LIN {X 0,Y 439.725,Z 495.084,A -85,B 0,C 180,E1 -9116.585,E2 -9116.585} C_VEL
LIN {X 0,Y 440.208,Z 487.996,A -85,B 0,C 180,E1 -9119.665,E2 -9119.665} C_VEL
LIN {X 0,Y 440.75,Z 482.421,A -85,B 0,C 180,E1 -9122.316,E2 -9122.316} C_VEL
LIN {X 0,Y 441.339,Z 477.409,A -85,B 0,C 180,E1 -9124.979,E2 -9124.979} C_VEL
LIN {X 0,Y 441.446,Z 473.772,A -85,B 0,C 180,E1 -9127.248,E2 -9127.248} C_VEL
LIN {X 0,Y 440.974,Z 470.762,A -85,B 0,C 180,E1 -9129.606,E2 -9129.606} C_VEL
LIN {X 0,Y 440.555,Z 468.312,A -85,B 0,C 180,E1 -9132.068,E2 -9132.068} C_VEL
LIN {X 0,Y 440.223,Z 466.544,A -85,B 0,C 180,E1 -9134.624,E2 -9134.624} C_VEL
LIN {X 0,Y 440.026,Z 465.358,A -85,B 0,C 180,E1 -9137.87,E2 -9137.87} C_VEL
LIN {X 0,Y 439.939,Z 465.185,A -85,B 0,C 180,E1 -9140.283,E2 -9140.283} C_VEL
LIN {X 0,Y 439.949,Z 465.547,A -85,B 0,C 180,E1 -9143.009,E2 -9143.009} C_VEL
LIN {X 0,Y 439.921,Z 466.128,A -85,B 0,C 180,E1 -9144.892,E2 -9144.892} C_VEL
LIN {X 0,Y 439.676,Z 467.615,A -85,B 0,C 180,E1 -9148.164,E2 -9148.164} C_VEL
LIN {X 0,Y 439.382,Z 469.659,A -85,B 0,C 180,E1 -9151.611,E2 -9151.611} C_VEL
LIN {X 0,Y 439.159,Z 471.579,A -85,B 0,C 180,E1 -9154.4,E2 -9154.4} C_VEL
LIN {X 0,Y 438.986,Z 473.84,A -85,B 0,C 180,E1 -9157.404,E2 -9157.404} C_VEL
LIN {X 0,Y 438.856,Z 476.233,A -85,B 0,C 180,E1 -9160.348,E2 -9160.348} C_VEL
LIN {X 0,Y 438.8,Z 479.014,A -85,B 0,C 180,E1 -9163.564,E2 -9163.564} C_VEL
LIN {X 0,Y 442.176,Z 491.192,A -85,B 0,C 180,E1 -9164.187,E2 -9164.187} C_VEL
LIN {X 0,Y 443.053,Z 496.365,A -85,B 0,C 180,E1 -9164.474,E2 -9164.474} C_VEL
LIN {X 0,Y 442.518,Z 508.604,A -85,B 0,C 180,E1 -9165.162,E2 -9165.162} C_VEL
LIN {X 0,Y 441.894,Z 520.706,A -85,B 0,C 180,E1 -9166.046,E2 -9166.046} C_VEL
LIN {X 0,Y 441.212,Z 532.256,A -85,B 0,C 180,E1 -9167.115,E2 -9167.115} C_VEL
LIN {X 0,Y 440.547,Z 542.238,A -85,B 0,C 180,E1 -9168.264,E2 -9168.264} C_VEL
LIN {X 0,Y 439.943,Z 551.84,A -85,B 0,C 180,E1 -9169.647,E2 -9169.647} C_VEL
LIN {X 0,Y 439.48,Z 559.568,A -85,B 0,C 180,E1 -9171.03,E2 -9171.03} C_VEL
LIN {X 0,Y 439.157,Z 564.797,A -85,B 0,C 180,E1 -9172.182,E2 -9172.182} C_VEL
LIN {X 0,Y 438.905,Z 569.893,A -85,B 0,C 180,E1 -9173.564,E2 -9173.564} C_VEL
LIN {X 0,Y 438.658,Z 573.844,A -85,B 0,C 180,E1 -9174.945,E2 -9174.945} C_VEL
LIN {X 0,Y 438.567,Z 576.739,A -85,B 0,C 180,E1 -9176.325,E2 -9176.325} C_VEL
LIN {X 0,Y 438.497,Z 578.115,A -85,B 0,C 180,E1 -9177.244,E2 -9177.244} C_VEL
LIN {X 0,Y 438.465,Z 579.07,A -85,B 0,C 180,E1 -9178.163,E2 -9178.163} C_VEL
LIN {X 0,Y 438.368,Z 579.638,A -85,B 0,C 180,E1 -9179.082,E2 -9179.082} C_VEL
LIN {X 0,Y 438.338,Z 579.807,A -85,B 0,C 180,E1 -9180,E2 -9180} C_VEL
LIN {X 0,Y 438.368,Z 579.532,A -85,B 0,C 180,E1 -9180.919,E2 -9180.919} C_VEL
LIN {X 0,Y 438.416,Z 578.858,A -85,B 0,C 180,E1 -9181.837,E2 -9181.837} C_VEL
LIN {X 0,Y 438.473,Z 577.791,A -85,B 0,C 180,E1 -9182.756,E2 -9182.756} C_VEL
LIN {X 0,Y 438.55,Z 576.305,A -85,B 0,C 180,E1 -9183.676,E2 -9183.676} C_VEL
LIN {X 0,Y 438.55,Z 573.247,A -85,B 0,C 180,E1 -9185.057,E2 -9185.057} C_VEL
LIN {X 0,Y 438.843,Z 569.115,A -85,B 0,C 180,E1 -9186.437,E2 -9186.437} C_VEL
LIN {X 0,Y 439.061,Z 562.782,A -85,B 0,C 180,E1 -9188.052,E2 -9188.052} C_VEL
LIN {X 0,Y 439.463,Z 555.889,A -85,B 0,C 180,E1 -9189.435,E2 -9189.435} C_VEL
LIN {X 0,Y 439.838,Z 548.87,A -85,B 0,C 180,E1 -9190.589,E2 -9190.589} C_VEL
LIN {X 0,Y 440.275,Z 540.435,A -85,B 0,C 180,E1 -9191.743,E2 -9191.743} C_VEL
LIN {X 0,Y 440.958,Z 530.059,A -85,B 0,C 180,E1 -9192.893,E2 -9192.893} C_VEL
LIN {X 0,Y 441.475,Z 518.456,A -85,B 0,C 180,E1 -9193.933,E2 -9193.933} C_VEL
LIN {X 0,Y 441.995,Z 507.041,A -85,B 0,C 180,E1 -9194.739,E2 -9194.739} C_VEL
LIN {X 0,Y 442.48,Z 495.475,A -85,B 0,C 180,E1 -9195.37,E2 -9195.37} C_VEL
LIN {X 0,Y 441.325,Z 488.815,A -85,B 0,C 180,E1 -9195.708,E2 -9195.708} C_VEL
LIN {X 0,Y 438.492,Z 476.161,A -85,B 0,C 180,E1 -9196.254,E2 -9196.254} C_VEL
LIN {X 0,Y 438.499,Z 472.466,A -85,B 0,C 180,E1 -9199.669,E2 -9199.669} C_VEL
LIN {X 0,Y 438.541,Z 469.335,A -85,B 0,C 180,E1 -9202.621,E2 -9202.621} C_VEL
LIN {X 0,Y 438.665,Z 465.591,A -85,B 0,C 180,E1 -9206.208,E2 -9206.208} C_VEL
LIN {X 0,Y 438.668,Z 463.019,A -85,B 0,C 180,E1 -9208.727,E2 -9208.727} C_VEL
LIN {X 0,Y 438.728,Z 461.844,A -85,B 0,C 180,E1 -9210.114,E2 -9210.114} C_VEL
LIN {X 0,Y 439.044,Z 461.798,A -85,B 0,C 180,E1 -9212.974,E2 -9212.974} C_VEL
LIN {X 0,Y 439.311,Z 461.762,A -85,B 0,C 180,E1 -9215.324,E2 -9215.324} C_VEL
LIN {X 0,Y 439.378,Z 461.756,A -85,B 0,C 180,E1 -9218.596,E2 -9218.596} C_VEL
LIN {X 0,Y 439.394,Z 461.749,A -85,B 0,C 180,E1 -9221.257,E2 -9221.257} C_VEL
LIN {X 0,Y 439.41,Z 461.75,A -85,B 0,C 180,E1 -9224.729,E2 -9224.729} C_VEL
LIN {X 0,Y 439.4,Z 461.753,A -85,B 0,C 180,E1 -9227.796,E2 -9227.796} C_VEL
LIN {X 0,Y 439.441,Z 461.747,A -85,B 0,C 180,E1 -9230.229,E2 -9230.229} C_VEL
LIN {X 0,Y 439.378,Z 461.753,A -85,B 0,C 180,E1 -9233.713,E2 -9233.713} C_VEL
LIN {X 0,Y 439.377,Z 461.754,A -85,B 0,C 180,E1 -9237.054,E2 -9237.054} C_VEL
LIN {X 0,Y 439.387,Z 461.753,A -85,B 0,C 180,E1 -9240.274,E2 -9240.274} C_VEL
LIN {X 0,Y 439.433,Z 461.747,A -85,B 0,C 180,E1 -9243.396,E2 -9243.396} C_VEL
LIN {X 0,Y 439.389,Z 461.753,A -85,B 0,C 180,E1 -9246.43,E2 -9246.43} C_VEL
LIN {X 0,Y 439.393,Z 461.752,A -85,B 0,C 180,E1 -9249.397,E2 -9249.397} C_VEL
LIN {X 0,Y 439.431,Z 461.748,A -85,B 0,C 180,E1 -9252.309,E2 -9252.309} C_VEL
LIN {X 0,Y 439.453,Z 461.744,A -85,B 0,C 180,E1 -9255.174,E2 -9255.174} C_VEL
LIN {X 0,Y 439.489,Z 461.742,A -85,B 0,C 180,E1 -9258.001,E2 -9258.001} C_VEL
LIN {X 0,Y 439.553,Z 461.735,A -85,B 0,C 180,E1 -9261.726,E2 -9261.726} C_VEL
LIN {X 0,Y 439.626,Z 461.724,A -85,B 0,C 180,E1 -9264.496,E2 -9264.496} C_VEL
LIN {X 0,Y 439.573,Z 461.729,A -85,B 0,C 180,E1 -9266.99,E2 -9266.99} C_VEL
LIN {X 0,Y 439.046,Z 461.796,A -85,B 0,C 180,E1 -9267.755,E2 -9267.755} C_VEL
LIN {X 0,Y 436.22,Z 462.147,A -85,B 0,C 180,E1 -9268.998,E2 -9268.998} C_VEL
LIN {X 0,Y 433.737,Z 462.459,A -85,B 0,C 180,E1 -9270.001,E2 -9270.001} C_VEL
LIN {X 0,Y 432.661,Z 462.589,A -85,B 0,C 180,E1 -9270.777,E2 -9270.777} C_VEL
LIN {X 0,Y 432.574,Z 462.599,A -85,B 0,C 180,E1 -9271.04,E2 -9271.04} C_VEL
LIN {X 0,Y 432.597,Z 462.597,A -85,B 0,C 180,E1 -9272.794,E2 -9272.794} C_VEL
LIN {X 0,Y 432.591,Z 462.602,A -85,B 0,C 180,E1 -9275.594,E2 -9275.594} C_VEL
LIN {X 0,Y 432.469,Z 462.617,A -85,B 0,C 180,E1 -9278.41,E2 -9278.41} C_VEL
LIN {X 0,Y 432.465,Z 462.617,A -85,B 0,C 180,E1 -9282.196,E2 -9282.196} C_VEL
LIN {X 0,Y 432.436,Z 462.62,A -85,B 0,C 180,E1 -9286.039,E2 -9286.039} C_VEL
LIN {X 0,Y 432.392,Z 462.626,A -85,B 0,C 180,E1 -9289.485,E2 -9289.485} C_VEL
LIN {X 0,Y 432.323,Z 462.632,A -85,B 0,C 180,E1 -9292.964,E2 -9292.964} C_VEL
LIN {X 0,Y 432.366,Z 462.629,A -85,B 0,C 180,E1 -9296.032,E2 -9296.032} C_VEL
LIN {X 0,Y 432.348,Z 462.629,A -85,B 0,C 180,E1 -9299.187,E2 -9299.187} C_VEL
LIN {X 0,Y 432.328,Z 462.633,A -85,B 0,C 180,E1 -9302.443,E2 -9302.443} C_VEL
LIN {X 0,Y 432.35,Z 462.63,A -85,B 0,C 180,E1 -9305.632,E2 -9305.632} C_VEL
LIN {X 0,Y 432.357,Z 462.625,A -85,B 0,C 180,E1 -9308.716,E2 -9308.716} C_VEL
LIN {X 0,Y 432.338,Z 462.632,A -85,B 0,C 180,E1 -9311.797,E2 -9311.797} C_VEL
LIN {X 0,Y 432.338,Z 462.632,A -85,B 0,C 180,E1 -9314.347,E2 -9314.347} C_VEL
LIN {X 0,Y 432.329,Z 462.632,A -85,B 0,C 180,E1 -9317.015,E2 -9317.015} C_VEL
LIN {X 0,Y 432.338,Z 462.634,A -85,B 0,C 180,E1 -9319.82,E2 -9319.82} C_VEL
LIN {X 0,Y 432.303,Z 462.634,A -85,B 0,C 180,E1 -9323.021,E2 -9323.021} C_VEL
LIN {X 0,Y 432.247,Z 462.645,A -85,B 0,C 180,E1 -9325.314,E2 -9325.314} C_VEL
LIN {X 0,Y 432.019,Z 462.674,A -85,B 0,C 180,E1 -9327.772,E2 -9327.772} C_VEL
LIN {X 0,Y 431.603,Z 462.726,A -85,B 0,C 180,E1 -9330.757,E2 -9330.757} C_VEL
LIN {X 0,Y 431.523,Z 462.84,A -85,B 0,C 180,E1 -9331.815,E2 -9331.815} C_VEL
LIN {X 0,Y 431.446,Z 466.378,A -85,B 0,C 180,E1 -9334.942,E2 -9334.942} C_VEL
LIN {X 0,Y 431.436,Z 470.05,A -85,B 0,C 180,E1 -9338.206,E2 -9338.206} C_VEL
LIN {X 0,Y 431.423,Z 473.199,A -85,B 0,C 180,E1 -9340.985,E2 -9340.985} C_VEL
LIN {X 0,Y 431.386,Z 476.277,A -85,B 0,C 180,E1 -9343.637,E2 -9343.637} C_VEL
LIN {X 0,Y 434.162,Z 488.766,A -85,B 0,C 180,E1 -9344.163,E2 -9344.163} C_VEL
LIN {X 0,Y 435.505,Z 496.504,A -85,B 0,C 180,E1 -9344.567,E2 -9344.567} C_VEL
LIN {X 0,Y 434.983,Z 508.593,A -85,B 0,C 180,E1 -9345.257,E2 -9345.257} C_VEL
LIN {X 0,Y 434.531,Z 519.197,A -85,B 0,C 180,E1 -9346.032,E2 -9346.032} C_VEL
LIN {X 0,Y 433.994,Z 529.992,A -85,B 0,C 180,E1 -9347.015,E2 -9347.015} C_VEL
LIN {X 0,Y 433.343,Z 539.442,A -85,B 0,C 180,E1 -9348.066,E2 -9348.066} C_VEL
LIN {X 0,Y 432.877,Z 548.128,A -85,B 0,C 180,E1 -9349.239,E2 -9349.239} C_VEL
LIN {X 0,Y 432.357,Z 556.622,A -85,B 0,C 180,E1 -9350.645,E2 -9350.645} C_VEL
LIN {X 0,Y 431.951,Z 563.423,A -85,B 0,C 180,E1 -9352.05,E2 -9352.05} C_VEL
LIN {X 0,Y 431.779,Z 568.864,A -85,B 0,C 180,E1 -9353.457,E2 -9353.457} C_VEL
LIN {X 0,Y 431.474,Z 573.12,A -85,B 0,C 180,E1 -9354.86,E2 -9354.86} C_VEL
LIN {X 0,Y 431.472,Z 576.287,A -85,B 0,C 180,E1 -9356.264,E2 -9356.264} C_VEL
LIN {X 0,Y 431.394,Z 577.87,A -85,B 0,C 180,E1 -9357.198,E2 -9357.198} C_VEL
LIN {X 0,Y 431.321,Z 578.99,A -85,B 0,C 180,E1 -9358.132,E2 -9358.132} C_VEL
LIN {X 0,Y 431.279,Z 580.034,A -85,B 0,C 180,E1 -9360,E2 -9360} C_VEL
LIN {X 0,Y 431.31,Z 579.937,A -85,B 0,C 180,E1 -9360.933,E2 -9360.933} C_VEL
LIN {X 0,Y 431.393,Z 579.41,A -85,B 0,C 180,E1 -9361.867,E2 -9361.867} C_VEL
LIN {X 0,Y 431.425,Z 578.499,A -85,B 0,C 180,E1 -9362.801,E2 -9362.801} C_VEL
LIN {X 0,Y 431.514,Z 577.184,A -85,B 0,C 180,E1 -9363.735,E2 -9363.735} C_VEL
LIN {X 0,Y 431.57,Z 574.377,A -85,B 0,C 180,E1 -9365.138,E2 -9365.138} C_VEL
LIN {X 0,Y 431.861,Z 570.513,A -85,B 0,C 180,E1 -9366.541,E2 -9366.541} C_VEL
LIN {X 0,Y 432.098,Z 565.493,A -85,B 0,C 180,E1 -9367.946,E2 -9367.946} C_VEL
LIN {X 0,Y 432.62,Z 557.957,A -85,B 0,C 180,E1 -9369.585,E2 -9369.585} C_VEL
LIN {X 0,Y 433.15,Z 549.779,A -85,B 0,C 180,E1 -9370.99,E2 -9370.99} C_VEL
LIN {X 0,Y 433.839,Z 539.573,A -85,B 0,C 180,E1 -9372.394,E2 -9372.394} C_VEL
LIN {X 0,Y 434.525,Z 529.567,A -85,B 0,C 180,E1 -9373.499,E2 -9373.499} C_VEL
LIN {X 0,Y 435.124,Z 518.422,A -85,B 0,C 180,E1 -9374.498,E2 -9374.498} C_VEL
LIN {X 0,Y 435.834,Z 506.924,A -85,B 0,C 180,E1 -9375.311,E2 -9375.311} C_VEL
LIN {X 0,Y 436.243,Z 496.479,A -85,B 0,C 180,E1 -9375.895,E2 -9375.895} C_VEL
LIN {X 0,Y 433.618,Z 485.375,A -85,B 0,C 180,E1 -9376.517,E2 -9376.517} C_VEL
LIN {X 0,Y 431.621,Z 478.702,A -85,B 0,C 180,E1 -9376.883,E2 -9376.883} C_VEL
LIN {X 0,Y 431.656,Z 475.198,A -85,B 0,C 180,E1 -9379.993,E2 -9379.993} C_VEL
LIN {X 0,Y 431.671,Z 471.756,A -85,B 0,C 180,E1 -9383.001,E2 -9383.001} C_VEL
LIN {X 0,Y 431.767,Z 467.645,A -85,B 0,C 180,E1 -9386.459,E2 -9386.459} C_VEL
LIN {X 0,Y 431.733,Z 464.394,A -85,B 0,C 180,E1 -9389.233,E2 -9389.233} C_VEL
LIN {X 0,Y 431.727,Z 462.935,A -85,B 0,C 180,E1 -9390.37,E2 -9390.37} C_VEL
LIN {X 0,Y 432.045,Z 462.672,A -85,B 0,C 180,E1 -9392.466,E2 -9392.466} C_VEL
LIN {X 0,Y 432.314,Z 462.636,A -85,B 0,C 180,E1 -9395.626,E2 -9395.626} C_VEL
LIN {X 0,Y 432.35,Z 462.63,A -85,B 0,C 180,E1 -9398.716,E2 -9398.716} C_VEL
LIN {X 0,Y 432.337,Z 462.632,A -85,B 0,C 180,E1 -9401.797,E2 -9401.797} C_VEL
LIN {X 0,Y 432.343,Z 462.633,A -85,B 0,C 180,E1 -9404.346,E2 -9404.346} C_VEL
LIN {X 0,Y 432.374,Z 462.673,A -85,B 0,C 180,E1 -9408.129,E2 -9408.129} C_VEL
LIN {X 0,Y 433.449,Z 468.757,A -85,B 0,C 180,E1 -9411.103,E2 -9411.103} C_VEL
LIN {X 0,Y 434.2,Z 473.235,A -85,B 0,C 180,E1 -9413.21,E2 -9413.21} C_VEL
LIN {X 0,Y 434.325,Z 477.103,A -85,B 0,C 180,E1 -9414.939,E2 -9414.939} C_VEL
LIN {X 0,Y 433.664,Z 484.792,A -85,B 0,C 180,E1 -9418.217,E2 -9418.217} C_VEL
LIN {X 0,Y 433.229,Z 491.9,A -85,B 0,C 180,E1 -9421.165,E2 -9421.165} C_VEL
LIN {X 0,Y 432.674,Z 500.183,A -85,B 0,C 180,E1 -9424.504,E2 -9424.504} C_VEL
LIN {X 0,Y 432.218,Z 509.175,A -85,B 0,C 180,E1 -9428.038,E2 -9428.038} C_VEL
LIN {X 0,Y 431.858,Z 518.157,A -85,B 0,C 180,E1 -9431.498,E2 -9431.498} C_VEL
LIN {X 0,Y 431.738,Z 523.3,A -85,B 0,C 180,E1 -9433.454,E2 -9433.454} C_VEL
LIN {X 0,Y 433.768,Z 537.812,A -85,B 0,C 180,E1 -9433.992,E2 -9433.992} C_VEL
LIN {X 0,Y 435.049,Z 549.897,A -85,B 0,C 180,E1 -9434.601,E2 -9434.601} C_VEL
LIN {X 0,Y 434.387,Z 562.251,A -85,B 0,C 180,E1 -9435.357,E2 -9435.357} C_VEL
LIN {X 0,Y 433.768,Z 573.811,A -85,B 0,C 180,E1 -9436.268,E2 -9436.268} C_VEL
LIN {X 0,Y 433.153,Z 584.686,A -85,B 0,C 180,E1 -9437.347,E2 -9437.347} C_VEL
LIN {X 0,Y 432.586,Z 594.309,A -85,B 0,C 180,E1 -9438.52,E2 -9438.52} C_VEL
LIN {X 0,Y 432.077,Z 602.225,A -85,B 0,C 180,E1 -9439.693,E2 -9439.693} C_VEL
LIN {X 0,Y 431.724,Z 609.974,A -85,B 0,C 180,E1 -9441.103,E2 -9441.103} C_VEL
LIN {X 0,Y 431.465,Z 616.192,A -85,B 0,C 180,E1 -9442.512,E2 -9442.512} C_VEL
LIN {X 0,Y 431.299,Z 621.368,A -85,B 0,C 180,E1 -9444.002,E2 -9444.002} C_VEL
LIN {X 0,Y 431.289,Z 624.889,A -85,B 0,C 180,E1 -9445.327,E2 -9445.327} C_VEL
LIN {X 0,Y 431.238,Z 626.819,A -85,B 0,C 180,E1 -9446.262,E2 -9446.262} C_VEL
LIN {X 0,Y 431.318,Z 628.308,A -85,B 0,C 180,E1 -9447.198,E2 -9447.198} C_VEL
LIN {X 0,Y 431.285,Z 629.327,A -85,B 0,C 180,E1 -9448.132,E2 -9448.132} C_VEL
LIN {X 0,Y 431.289,Z 629.944,A -85,B 0,C 180,E1 -9449.066,E2 -9449.066} C_VEL
LIN {X 0,Y 431.277,Z 630.156,A -85,B 0,C 180,E1 -9450,E2 -9450} C_VEL
LIN {X 0,Y 431.276,Z 629.931,A -85,B 0,C 180,E1 -9450.934,E2 -9450.934} C_VEL
LIN {X 0,Y 431.287,Z 629.272,A -85,B 0,C 180,E1 -9451.868,E2 -9451.868} C_VEL
LIN {X 0,Y 431.326,Z 628.209,A -85,B 0,C 180,E1 -9452.802,E2 -9452.802} C_VEL
LIN {X 0,Y 431.245,Z 626.725,A -85,B 0,C 180,E1 -9453.738,E2 -9453.738} C_VEL
LIN {X 0,Y 431.329,Z 623.63,A -85,B 0,C 180,E1 -9455.142,E2 -9455.142} C_VEL
LIN {X 0,Y 431.376,Z 619.459,A -85,B 0,C 180,E1 -9456.549,E2 -9456.549} C_VEL
LIN {X 0,Y 431.6,Z 613.079,A -85,B 0,C 180,E1 -9458.191,E2 -9458.191} C_VEL
LIN {X 0,Y 431.891,Z 606.139,A -85,B 0,C 180,E1 -9459.602,E2 -9459.602} C_VEL
LIN {X 0,Y 432.365,Z 597.585,A -85,B 0,C 180,E1 -9461.011,E2 -9461.011} C_VEL
LIN {X 0,Y 432.9,Z 588.865,A -85,B 0,C 180,E1 -9462.184,E2 -9462.184} C_VEL
LIN {X 0,Y 433.491,Z 578.875,A -85,B 0,C 180,E1 -9463.292,E2 -9463.292} C_VEL
LIN {X 0,Y 434.191,Z 567.869,A -85,B 0,C 180,E1 -9464.291,E2 -9464.291} C_VEL
LIN {X 0,Y 434.922,Z 556.771,A -85,B 0,C 180,E1 -9465.104,E2 -9465.104} C_VEL
LIN {X 0,Y 435.135,Z 547.972,A -85,B 0,C 180,E1 -9465.636,E2 -9465.636} C_VEL
LIN {X 0,Y 433.873,Z 534.203,A -85,B 0,C 180,E1 -9466.359,E2 -9466.359} C_VEL
LIN {X 0,Y 431.663,Z 520.58,A -85,B 0,C 180,E1 -9466.942,E2 -9466.942} C_VEL
LIN {X 0,Y 431.956,Z 511.211,A -85,B 0,C 180,E1 -9470.476,E2 -9470.476} C_VEL
LIN {X 0,Y 432.235,Z 503.577,A -85,B 0,C 180,E1 -9473.476,E2 -9473.476} C_VEL
LIN {X 0,Y 432.696,Z 495.781,A -85,B 0,C 180,E1 -9476.705,E2 -9476.705} C_VEL
LIN {X 0,Y 433.19,Z 489.162,A -85,B 0,C 180,E1 -9479.658,E2 -9479.658} C_VEL
LIN {X 0,Y 433.75,Z 483.692,A -85,B 0,C 180,E1 -9482.323,E2 -9482.323} C_VEL
LIN {X 0,Y 434.28,Z 479.633,A -85,B 0,C 180,E1 -9484.5,E2 -9484.5} C_VEL
LIN {X 0,Y 434.482,Z 475.964,A -85,B 0,C 180,E1 -9486.762,E2 -9486.762} C_VEL
LIN {X 0,Y 434.141,Z 472.803,A -85,B 0,C 180,E1 -9489.15,E2 -9489.15} C_VEL
LIN {X 0,Y 433.676,Z 470.093,A -85,B 0,C 180,E1 -9491.801,E2 -9491.801} C_VEL
LIN {X 0,Y 433.307,Z 468.189,A -85,B 0,C 180,E1 -9494.467,E2 -9494.467} C_VEL
LIN {X 0,Y 433.135,Z 467.082,A -85,B 0,C 180,E1 -9497.04,E2 -9497.04} C_VEL
LIN {X 0,Y 432.998,Z 466.649,A -85,B 0,C 180,E1 -9499.717,E2 -9499.717} C_VEL
LIN {X 0,Y 432.987,Z 466.95,A -85,B 0,C 180,E1 -9503.09,E2 -9503.09} C_VEL
LIN {X 0,Y 432.852,Z 467.822,A -85,B 0,C 180,E1 -9505.901,E2 -9505.901} C_VEL
LIN {X 0,Y 432.637,Z 469.107,A -85,B 0,C 180,E1 -9508.679,E2 -9508.679} C_VEL
LIN {X 0,Y 432.334,Z 470.952,A -85,B 0,C 180,E1 -9511.873,E2 -9511.873} C_VEL
LIN {X 0,Y 432.116,Z 473.054,A -85,B 0,C 180,E1 -9514.984,E2 -9514.984} C_VEL
LIN {X 0,Y 431.942,Z 475.336,A -85,B 0,C 180,E1 -9518.038,E2 -9518.038} C_VEL
LIN {X 0,Y 431.869,Z 477.718,A -85,B 0,C 180,E1 -9521.006,E2 -9521.006} C_VEL
LIN {X 0,Y 431.796,Z 479.791,A -85,B 0,C 180,E1 -9523.228,E2 -9523.228} C_VEL
LIN {X 0,Y 435.363,Z 492.152,A -85,B 0,C 180,E1 -9523.9,E2 -9523.9} C_VEL
LIN {X 0,Y 436.316,Z 497.847,A -85,B 0,C 180,E1 -9524.228,E2 -9524.228} C_VEL
LIN {X 0,Y 435.766,Z 509.831,A -85,B 0,C 180,E1 -9524.926,E2 -9524.926} C_VEL
LIN {X 0,Y 435.076,Z 521.704,A -85,B 0,C 180,E1 -9525.822,E2 -9525.822} C_VEL
LIN {X 0,Y 434.341,Z 533.084,A -85,B 0,C 180,E1 -9526.907,E2 -9526.907} C_VEL
LIN {X 0,Y 433.634,Z 542.93,A -85,B 0,C 180,E1 -9528.075,E2 -9528.075} C_VEL
LIN {X 0,Y 432.986,Z 552.482,A -85,B 0,C 180,E1 -9529.479,E2 -9529.479} C_VEL
LIN {X 0,Y 432.502,Z 560.172,A -85,B 0,C 180,E1 -9530.884,E2 -9530.884} C_VEL
LIN {X 0,Y 432.004,Z 567.193,A -85,B 0,C 180,E1 -9532.522,E2 -9532.522} C_VEL
LIN {X 0,Y 431.74,Z 571.862,A -85,B 0,C 180,E1 -9533.926,E2 -9533.926} C_VEL
LIN {X 0,Y 431.63,Z 575.41,A -85,B 0,C 180,E1 -9535.33,E2 -9535.33} C_VEL
LIN {X 0,Y 431.516,Z 577.232,A -85,B 0,C 180,E1 -9536.265,E2 -9536.265} C_VEL
LIN {X 0,Y 431.425,Z 578.584,A -85,B 0,C 180,E1 -9537.199,E2 -9537.199} C_VEL
LIN {X 0,Y 431.409,Z 579.522,A -85,B 0,C 180,E1 -9538.133,E2 -9538.133} C_VEL
LIN {X 0,Y 431.31,Z 580.076,A -85,B 0,C 180,E1 -9539.067,E2 -9539.067} C_VEL
LIN {X 0,Y 431.278,Z 580.227,A -85,B 0,C 180,E1 -9540,E2 -9540} C_VEL
LIN {X 0,Y 431.292,Z 579.934,A -85,B 0,C 180,E1 -9540.934,E2 -9540.934} C_VEL
LIN {X 0,Y 431.334,Z 579.244,A -85,B 0,C 180,E1 -9541.868,E2 -9541.868} C_VEL
LIN {X 0,Y 431.403,Z 578.161,A -85,B 0,C 180,E1 -9542.802,E2 -9542.802} C_VEL
LIN {X 0,Y 431.473,Z 576.648,A -85,B 0,C 180,E1 -9543.736,E2 -9543.736} C_VEL
LIN {X 0,Y 431.485,Z 573.556,A -85,B 0,C 180,E1 -9545.14,E2 -9545.14} C_VEL
LIN {X 0,Y 431.785,Z 569.382,A -85,B 0,C 180,E1 -9546.543,E2 -9546.543} C_VEL
LIN {X 0,Y 432.011,Z 562.998,A -85,B 0,C 180,E1 -9548.184,E2 -9548.184} C_VEL
LIN {X 0,Y 432.455,Z 556.058,A -85,B 0,C 180,E1 -9549.589,E2 -9549.589} C_VEL
LIN {X 0,Y 432.86,Z 548.987,A -85,B 0,C 180,E1 -9550.762,E2 -9550.762} C_VEL
LIN {X 0,Y 433.304,Z 540.485,A -85,B 0,C 180,E1 -9551.935,E2 -9551.935} C_VEL
LIN {X 0,Y 434.031,Z 530.023,A -85,B 0,C 180,E1 -9553.103,E2 -9553.103} C_VEL
LIN {X 0,Y 434.581,Z 518.343,A -85,B 0,C 180,E1 -9554.159,E2 -9554.159} C_VEL
LIN {X 0,Y 435.138,Z 506.769,A -85,B 0,C 180,E1 -9554.977,E2 -9554.977} C_VEL
LIN {X 0,Y 435.504,Z 495.064,A -85,B 0,C 180,E1 -9555.623,E2 -9555.623} C_VEL
LIN {X 0,Y 432.548,Z 481.624,A -85,B 0,C 180,E1 -9556.281,E2 -9556.281} C_VEL
LIN {X 0,Y 431.414,Z 476.484,A -85,B 0,C 180,E1 -9556.504,E2 -9556.504} C_VEL
LIN {X 0,Y 431.42,Z 472.725,A -85,B 0,C 180,E1 -9560.005,E2 -9560.005} C_VEL
LIN {X 0,Y 431.498,Z 469.551,A -85,B 0,C 180,E1 -9563.011,E2 -9563.011} C_VEL
LIN {X 0,Y 431.602,Z 466.032,A -85,B 0,C 180,E1 -9566.415,E2 -9566.415} C_VEL
LIN {X 0,Y 431.614,Z 463.167,A -85,B 0,C 180,E1 -9569.242,E2 -9569.242} C_VEL
LIN {X 0,Y 431.704,Z 462.718,A -85,B 0,C 180,E1 -9570.365,E2 -9570.365} C_VEL
LIN {X 0,Y 432.06,Z 462.667,A -85,B 0,C 180,E1 -9573.577,E2 -9573.577} C_VEL
LIN {X 0,Y 432.27,Z 462.64,A -85,B 0,C 180,E1 -9575.825,E2 -9575.825} C_VEL
LIN {X 0,Y 432.341,Z 462.632,A -85,B 0,C 180,E1 -9578.714,E2 -9578.714} C_VEL
LIN {X 0,Y 432.339,Z 462.63,A -85,B 0,C 180,E1 -9581.797,E2 -9581.797} C_VEL
LIN {X 0,Y 432.345,Z 462.631,A -85,B 0,C 180,E1 -9584.347,E2 -9584.347} C_VEL
LIN {X 0,Y 432.324,Z 462.633,A -85,B 0,C 180,E1 -9587.016,E2 -9587.016} C_VEL
LIN {X 0,Y 432.345,Z 462.63,A -85,B 0,C 180,E1 -9589.82,E2 -9589.82} C_VEL
LIN {X 0,Y 432.315,Z 462.631,A -85,B 0,C 180,E1 -9593.023,E2 -9593.023} C_VEL
LIN {X 0,Y 432.364,Z 462.631,A -85,B 0,C 180,E1 -9595.997,E2 -9595.997} C_VEL
LIN {X 0,Y 432.352,Z 462.63,A -85,B 0,C 180,E1 -9599.49,E2 -9599.49} C_VEL
LIN {X 0,Y 432.395,Z 462.623,A -85,B 0,C 180,E1 -9602.928,E2 -9602.928} C_VEL
LIN {X 0,Y 432.373,Z 462.629,A -85,B 0,C 180,E1 -9606.023,E2 -9606.023} C_VEL
LIN {X 0,Y 432.355,Z 462.628,A -85,B 0,C 180,E1 -9609.046,E2 -9609.046} C_VEL
LIN {X 0,Y 432.379,Z 462.626,A -85,B 0,C 180,E1 -9612.011,E2 -9612.011} C_VEL
LIN {X 0,Y 432.401,Z 462.623,A -85,B 0,C 180,E1 -9614.927,E2 -9614.927} C_VEL
LIN {X 0,Y 432.465,Z 462.616,A -85,B 0,C 180,E1 -9617.804,E2 -9617.804} C_VEL
LIN {X 0,Y 432.497,Z 462.612,A -85,B 0,C 180,E1 -9621.59,E2 -9621.59} C_VEL
LIN {X 0,Y 432.602,Z 462.599,A -85,B 0,C 180,E1 -9624.406,E2 -9624.406} C_VEL
LIN {X 0,Y 432.609,Z 462.599,A -85,B 0,C 180,E1 -9628.138,E2 -9628.138} C_VEL
LIN {X 0,Y 432.738,Z 462.584,A -85,B 0,C 180,E1 -9630,E2 -9630} C_VEL
LIN {X 0,Y 432.574,Z 462.599,A -85,B 0,C 180,E1 -9631.04,E2 -9631.04} C_VEL
LIN {X 0,Y 431.875,Z 462.691,A -85,B 0,C 180,E1 -9631.817,E2 -9631.817} C_VEL
LIN {X 0,Y 428.911,Z 463.056,A -85,B 0,C 180,E1 -9633.076,E2 -9633.076} C_VEL
LIN {X 0,Y 426.456,Z 463.365,A -85,B 0,C 180,E1 -9634.093,E2 -9634.093} C_VEL
LIN {X 0,Y 425.473,Z 463.485,A -85,B 0,C 180,E1 -9634.88,E2 -9634.88} C_VEL
LIN {X 0,Y 425.432,Z 463.49,A -85,B 0,C 180,E1 -9635.147,E2 -9635.147} C_VEL
LIN {X 0,Y 425.484,Z 463.486,A -85,B 0,C 180,E1 -9637.663,E2 -9637.663} C_VEL
LIN {X 0,Y 425.37,Z 463.5,A -85,B 0,C 180,E1 -9640.471,E2 -9640.471} C_VEL
LIN {X 0,Y 425.371,Z 463.497,A -85,B 0,C 180,E1 -9643.374,E2 -9643.374} C_VEL
LIN {X 0,Y 425.367,Z 463.499,A -85,B 0,C 180,E1 -9646.605,E2 -9646.605} C_VEL
LIN {X 0,Y 425.334,Z 463.505,A -85,B 0,C 180,E1 -9649.636,E2 -9649.636} C_VEL
LIN {X 0,Y 425.293,Z 463.51,A -85,B 0,C 180,E1 -9652.339,E2 -9652.339} C_VEL
LIN {X 0,Y 425.296,Z 463.508,A -85,B 0,C 180,E1 -9655.445,E2 -9655.445} C_VEL
LIN {X 0,Y 425.353,Z 463.502,A -85,B 0,C 180,E1 -9657.558,E2 -9657.558} C_VEL
LIN {X 0,Y 425.293,Z 463.508,A -85,B 0,C 180,E1 -9660.816,E2 -9660.816} C_VEL
LIN {X 0,Y 425.317,Z 463.507,A -85,B 0,C 180,E1 -9664.288,E2 -9664.288} C_VEL
LIN {X 0,Y 425.29,Z 463.511,A -85,B 0,C 180,E1 -9667.693,E2 -9667.693} C_VEL
LIN {X 0,Y 425.288,Z 463.508,A -85,B 0,C 180,E1 -9670.521,E2 -9670.521} C_VEL
LIN {X 0,Y 425.262,Z 463.514,A -85,B 0,C 180,E1 -9673.351,E2 -9673.351} C_VEL
LIN {X 0,Y 425.268,Z 463.511,A -85,B 0,C 180,E1 -9676.648,E2 -9676.648} C_VEL
LIN {X 0,Y 425.291,Z 463.512,A -85,B 0,C 180,E1 -9679.873,E2 -9679.873} C_VEL
LIN {X 0,Y 425.278,Z 463.508,A -85,B 0,C 180,E1 -9682.489,E2 -9682.489} C_VEL
LIN {X 0,Y 425.253,Z 463.513,A -85,B 0,C 180,E1 -9684.659,E2 -9684.659} C_VEL
LIN {X 0,Y 425.003,Z 463.548,A -85,B 0,C 180,E1 -9687.496,E2 -9687.496} C_VEL
LIN {X 0,Y 424.507,Z 463.612,A -85,B 0,C 180,E1 -9691.337,E2 -9691.337} C_VEL
LIN {X 0,Y 424.444,Z 464.092,A -85,B 0,C 180,E1 -9692.378,E2 -9692.378} C_VEL
LIN {X 0,Y 424.384,Z 467.734,A -85,B 0,C 180,E1 -9695.62,E2 -9695.62} C_VEL
LIN {X 0,Y 424.353,Z 471.148,A -85,B 0,C 180,E1 -9698.632,E2 -9698.632} C_VEL
LIN {X 0,Y 424.313,Z 474.565,A -85,B 0,C 180,E1 -9701.657,E2 -9701.657} C_VEL
LIN {X 0,Y 424.302,Z 476.555,A -85,B 0,C 180,E1 -9703.402,E2 -9703.402} C_VEL
LIN {X 0,Y 426.964,Z 488.726,A -85,B 0,C 180,E1 -9703.92,E2 -9703.92} C_VEL
LIN {X 0,Y 428.608,Z 497.055,A -85,B 0,C 180,E1 -9704.366,E2 -9704.366} C_VEL
LIN {X 0,Y 428.025,Z 510.097,A -85,B 0,C 180,E1 -9705.134,E2 -9705.134} C_VEL
LIN {X 0,Y 427.46,Z 521.914,A -85,B 0,C 180,E1 -9706.049,E2 -9706.049} C_VEL
LIN {X 0,Y 426.819,Z 533.31,A -85,B 0,C 180,E1 -9707.156,E2 -9707.156} C_VEL
LIN {X 0,Y 426.162,Z 543.138,A -85,B 0,C 180,E1 -9708.345,E2 -9708.345} C_VEL
LIN {X 0,Y 425.578,Z 552.713,A -85,B 0,C 180,E1 -9709.774,E2 -9709.774} C_VEL
LIN {X 0,Y 425.1,Z 560.367,A -85,B 0,C 180,E1 -9711.203,E2 -9711.203} C_VEL
LIN {X 0,Y 424.723,Z 567.606,A -85,B 0,C 180,E1 -9712.918,E2 -9712.918} C_VEL
LIN {X 0,Y 424.535,Z 572.108,A -85,B 0,C 180,E1 -9714.299,E2 -9714.299} C_VEL
LIN {X 0,Y 424.389,Z 575.67,A -85,B 0,C 180,E1 -9715.726,E2 -9715.726} C_VEL
LIN {X 0,Y 424.327,Z 578.207,A -85,B 0,C 180,E1 -9717.152,E2 -9717.152} C_VEL
LIN {X 0,Y 424.242,Z 579.357,A -85,B 0,C 180,E1 -9718.101,E2 -9718.101} C_VEL
LIN {X 0,Y 424.204,Z 580.439,A -85,B 0,C 180,E1 -9720,E2 -9720} C_VEL
LIN {X 0,Y 424.237,Z 580.374,A -85,B 0,C 180,E1 -9720.949,E2 -9720.949} C_VEL
LIN {X 0,Y 424.309,Z 579.865,A -85,B 0,C 180,E1 -9721.898,E2 -9721.898} C_VEL
LIN {X 0,Y 424.462,Z 577.671,A -85,B 0,C 180,E1 -9723.797,E2 -9723.797} C_VEL
LIN {X 0,Y 424.503,Z 574.89,A -85,B 0,C 180,E1 -9725.224,E2 -9725.224} C_VEL
LIN {X 0,Y 424.825,Z 571.051,A -85,B 0,C 180,E1 -9726.65,E2 -9726.65} C_VEL
LIN {X 0,Y 425.107,Z 566.055,A -85,B 0,C 180,E1 -9728.078,E2 -9728.078} C_VEL
LIN {X 0,Y 425.656,Z 558.579,A -85,B 0,C 180,E1 -9729.743,E2 -9729.743} C_VEL
LIN {X 0,Y 426.217,Z 550.502,A -85,B 0,C 180,E1 -9731.171,E2 -9731.171} C_VEL
LIN {X 0,Y 426.739,Z 542.231,A -85,B 0,C 180,E1 -9732.362,E2 -9732.362} C_VEL
LIN {X 0,Y 427.548,Z 532.495,A -85,B 0,C 180,E1 -9733.507,E2 -9733.507} C_VEL
LIN {X 0,Y 428.192,Z 522.801,A -85,B 0,C 180,E1 -9734.446,E2 -9734.446} C_VEL
LIN {X 0,Y 428.87,Z 511.599,A -85,B 0,C 180,E1 -9735.322,E2 -9735.322} C_VEL
LIN {X 0,Y 429.585,Z 498.012,A -85,B 0,C 180,E1 -9736.148,E2 -9736.148} C_VEL
LIN {X 0,Y 426.924,Z 486.798,A -85,B 0,C 180,E1 -9736.822,E2 -9736.822} C_VEL
LIN {X 0,Y 424.598,Z 479.229,A -85,B 0,C 180,E1 -9737.242,E2 -9737.242} C_VEL
LIN {X 0,Y 424.604,Z 475.772,A -85,B 0,C 180,E1 -9740.34,E2 -9740.34} C_VEL
LIN {X 0,Y 424.66,Z 472.309,A -85,B 0,C 180,E1 -9743.403,E2 -9743.403} C_VEL
LIN {X 0,Y 424.753,Z 468.513,A -85,B 0,C 180,E1 -9746.685,E2 -9746.685} C_VEL
LIN {X 0,Y 424.721,Z 464.808,A -85,B 0,C 180,E1 -9749.763,E2 -9749.763} C_VEL
LIN {X 0,Y 424.732,Z 463.582,A -85,B 0,C 180,E1 -9750.861,E2 -9750.861} C_VEL
LIN {X 0,Y 425.065,Z 463.541,A -85,B 0,C 180,E1 -9753.067,E2 -9753.067} C_VEL
LIN {X 0,Y 425.263,Z 463.515,A -85,B 0,C 180,E1 -9755.925,E2 -9755.925} C_VEL
LIN {X 0,Y 425.302,Z 463.508,A -85,B 0,C 180,E1 -9759.044,E2 -9759.044} C_VEL
LIN {X 0,Y 425.28,Z 463.512,A -85,B 0,C 180,E1 -9762.652,E2 -9762.652} C_VEL
LIN {X 0,Y 425.263,Z 463.515,A -85,B 0,C 180,E1 -9766.044,E2 -9766.044} C_VEL
LIN {X 0,Y 425.35,Z 463.671,A -85,B 0,C 180,E1 -9767.927,E2 -9767.927} C_VEL
LIN {X 0,Y 426.518,Z 470.319,A -85,B 0,C 180,E1 -9771.233,E2 -9771.233} C_VEL
LIN {X 0,Y 427.305,Z 475.515,A -85,B 0,C 180,E1 -9773.699,E2 -9773.699} C_VEL
LIN {X 0,Y 427.226,Z 479.171,A -85,B 0,C 180,E1 -9775.337,E2 -9775.337} C_VEL
LIN {X 0,Y 426.555,Z 487.55,A -85,B 0,C 180,E1 -9778.955,E2 -9778.955} C_VEL
LIN {X 0,Y 426.038,Z 494.719,A -85,B 0,C 180,E1 -9781.956,E2 -9781.956} C_VEL
LIN {X 0,Y 425.484,Z 502.907,A -85,B 0,C 180,E1 -9785.295,E2 -9785.295} C_VEL
LIN {X 0,Y 425.076,Z 511.356,A -85,B 0,C 180,E1 -9788.67,E2 -9788.67} C_VEL
LIN {X 0,Y 424.725,Z 520.311,A -85,B 0,C 180,E1 -9792.174,E2 -9792.174} C_VEL
LIN {X 0,Y 424.658,Z 522.666,A -85,B 0,C 180,E1 -9793.087,E2 -9793.087} C_VEL
LIN {X 0,Y 427.304,Z 542.644,A -85,B 0,C 180,E1 -9794.009,E2 -9794.009} C_VEL
LIN {X 0,Y 428.052,Z 550.918,A -85,B 0,C 180,E1 -9794.465,E2 -9794.465} C_VEL
LIN {X 0,Y 427.372,Z 562.953,A -85,B 0,C 180,E1 -9795.233,E2 -9795.233} C_VEL
LIN {X 0,Y 426.727,Z 574.262,A -85,B 0,C 180,E1 -9796.162,E2 -9796.162} C_VEL
LIN {X 0,Y 426.116,Z 584.962,A -85,B 0,C 180,E1 -9797.256,E2 -9797.256} C_VEL
LIN {X 0,Y 425.59,Z 593.581,A -85,B 0,C 180,E1 -9798.329,E2 -9798.329} C_VEL
LIN {X 0,Y 425.049,Z 601.551,A -85,B 0,C 180,E1 -9799.521,E2 -9799.521} C_VEL
LIN {X 0,Y 424.658,Z 609.368,A -85,B 0,C 180,E1 -9800.954,E2 -9800.954} C_VEL
LIN {X 0,Y 424.385,Z 615.628,A -85,B 0,C 180,E1 -9802.387,E2 -9802.387} C_VEL
LIN {X 0,Y 424.279,Z 620.098,A -85,B 0,C 180,E1 -9803.656,E2 -9803.656} C_VEL
LIN {X 0,Y 424.223,Z 624.394,A -85,B 0,C 180,E1 -9805.249,E2 -9805.249} C_VEL
LIN {X 0,Y 424.147,Z 626.337,A -85,B 0,C 180,E1 -9806.2,E2 -9806.2} C_VEL
LIN {X 0,Y 424.246,Z 627.851,A -85,B 0,C 180,E1 -9807.151,E2 -9807.151} C_VEL
LIN {X 0,Y 424.207,Z 628.884,A -85,B 0,C 180,E1 -9808.101,E2 -9808.101} C_VEL
LIN {X 0,Y 424.202,Z 629.509,A -85,B 0,C 180,E1 -9809.051,E2 -9809.051} C_VEL
LIN {X 0,Y 424.218,Z 629.731,A -85,B 0,C 180,E1 -9810,E2 -9810} C_VEL
LIN {X 0,Y 424.19,Z 629.522,A -85,B 0,C 180,E1 -9810.949,E2 -9810.949} C_VEL
LIN {X 0,Y 424.209,Z 628.869,A -85,B 0,C 180,E1 -9811.899,E2 -9811.899} C_VEL
LIN {X 0,Y 424.235,Z 627.81,A -85,B 0,C 180,E1 -9812.849,E2 -9812.849} C_VEL
LIN {X 0,Y 424.152,Z 626.331,A -85,B 0,C 180,E1 -9813.8,E2 -9813.8} C_VEL
LIN {X 0,Y 424.237,Z 623.249,A -85,B 0,C 180,E1 -9815.228,E2 -9815.228} C_VEL
LIN {X 0,Y 424.299,Z 619.09,A -85,B 0,C 180,E1 -9816.658,E2 -9816.658} C_VEL
LIN {X 0,Y 424.532,Z 612.737,A -85,B 0,C 180,E1 -9818.329,E2 -9818.329} C_VEL
LIN {X 0,Y 424.853,Z 605.827,A -85,B 0,C 180,E1 -9819.762,E2 -9819.762} C_VEL
LIN {X 0,Y 425.376,Z 597.309,A -85,B 0,C 180,E1 -9821.194,E2 -9821.194} C_VEL
LIN {X 0,Y 425.887,Z 588.659,A -85,B 0,C 180,E1 -9822.388,E2 -9822.388} C_VEL
LIN {X 0,Y 426.594,Z 578.013,A -85,B 0,C 180,E1 -9823.588,E2 -9823.588} C_VEL
LIN {X 0,Y 427.428,Z 566.466,A -85,B 0,C 180,E1 -9824.644,E2 -9824.644} C_VEL
LIN {X 0,Y 428.197,Z 555.161,A -85,B 0,C 180,E1 -9825.469,E2 -9825.469} C_VEL
LIN {X 0,Y 428.266,Z 548.38,A -85,B 0,C 180,E1 -9825.893,E2 -9825.893} C_VEL
LIN {X 0,Y 427.013,Z 534.488,A -85,B 0,C 180,E1 -9826.661,E2 -9826.661} C_VEL
LIN {X 0,Y 424.953,Z 522.186,A -85,B 0,C 180,E1 -9827.215,E2 -9827.215} C_VEL
LIN {X 0,Y 424.635,Z 519.993,A -85,B 0,C 180,E1 -9827.332,E2 -9827.332} C_VEL
LIN {X 0,Y 424.921,Z 510.95,A -85,B 0,C 180,E1 -9830.83,E2 -9830.83} C_VEL
LIN {X 0,Y 425.304,Z 502.16,A -85,B 0,C 180,E1 -9834.401,E2 -9834.401} C_VEL
LIN {X 0,Y 425.827,Z 494.923,A -85,B 0,C 180,E1 -9837.524,E2 -9837.524} C_VEL
LIN {X 0,Y 426.492,Z 487.496,A -85,B 0,C 180,E1 -9841.031,E2 -9841.031} C_VEL
LIN {X 0,Y 427.197,Z 481.859,A -85,B 0,C 180,E1 -9844.011,E2 -9844.011} C_VEL
LIN {X 0,Y 427.529,Z 478.04,A -85,B 0,C 180,E1 -9846.342,E2 -9846.342} C_VEL
LIN {X 0,Y 427.305,Z 474.87,A -85,B 0,C 180,E1 -9848.682,E2 -9848.682} C_VEL
LIN {X 0,Y 426.819,Z 472.197,A -85,B 0,C 180,E1 -9851.196,E2 -9851.196} C_VEL
LIN {X 0,Y 426.465,Z 470.149,A -85,B 0,C 180,E1 -9853.8,E2 -9853.8} C_VEL
LIN {X 0,Y 426.243,Z 468.783,A -85,B 0,C 180,E1 -9856.509,E2 -9856.509} C_VEL
LIN {X 0,Y 426.057,Z 468.151,A -85,B 0,C 180,E1 -9859.358,E2 -9859.358} C_VEL
LIN {X 0,Y 426.037,Z 468.222,A -85,B 0,C 180,E1 -9862.384,E2 -9862.384} C_VEL
LIN {X 0,Y 425.949,Z 468.743,A -85,B 0,C 180,E1 -9864.726,E2 -9864.726} C_VEL
LIN {X 0,Y 425.681,Z 470.062,A -85,B 0,C 180,E1 -9868.108,E2 -9868.108} C_VEL
LIN {X 0,Y 425.393,Z 471.802,A -85,B 0,C 180,E1 -9871.372,E2 -9871.372} C_VEL
LIN {X 0,Y 425.104,Z 473.831,A -85,B 0,C 180,E1 -9874.542,E2 -9874.542} C_VEL
LIN {X 0,Y 424.919,Z 476.202,A -85,B 0,C 180,E1 -9877.853,E2 -9877.853} C_VEL
LIN {X 0,Y 424.83,Z 478.404,A -85,B 0,C 180,E1 -9880.679,E2 -9880.679} C_VEL
LIN {X 0,Y 424.737,Z 480.197,A -85,B 0,C 180,E1 -9882.841,E2 -9882.841} C_VEL
LIN {X 0,Y 428.594,Z 493.148,A -85,B 0,C 180,E1 -9883.593,E2 -9883.593} C_VEL
LIN {X 0,Y 429.633,Z 498.308,A -85,B 0,C 180,E1 -9883.915,E2 -9883.915} C_VEL
LIN {X 0,Y 429,Z 511.045,A -85,B 0,C 180,E1 -9884.683,E2 -9884.683} C_VEL
LIN {X 0,Y 428.267,Z 522.726,A -85,B 0,C 180,E1 -9885.592,E2 -9885.592} C_VEL
LIN {X 0,Y 427.488,Z 534.006,A -85,B 0,C 180,E1 -9886.693,E2 -9886.693} C_VEL
LIN {X 0,Y 426.759,Z 543.75,A -85,B 0,C 180,E1 -9887.879,E2 -9887.879} C_VEL
LIN {X 0,Y 426.044,Z 553.209,A -85,B 0,C 180,E1 -9889.305,E2 -9889.305} C_VEL
LIN {X 0,Y 425.532,Z 560.801,A -85,B 0,C 180,E1 -9890.734,E2 -9890.734} C_VEL
LIN {X 0,Y 424.992,Z 567.772,A -85,B 0,C 180,E1 -9892.398,E2 -9892.398} C_VEL
LIN {X 0,Y 424.709,Z 572.416,A -85,B 0,C 180,E1 -9893.825,E2 -9893.825} C_VEL
LIN {X 0,Y 424.568,Z 575.939,A -85,B 0,C 180,E1 -9895.253,E2 -9895.253} C_VEL
LIN {X 0,Y 424.465,Z 577.741,A -85,B 0,C 180,E1 -9896.203,E2 -9896.203} C_VEL
LIN {X 0,Y 424.357,Z 579.072,A -85,B 0,C 180,E1 -9897.152,E2 -9897.152} C_VEL
LIN {X 0,Y 424.338,Z 579.994,A -85,B 0,C 180,E1 -9898.102,E2 -9898.102} C_VEL
LIN {X 0,Y 424.254,Z 580.529,A -85,B 0,C 180,E1 -9899.051,E2 -9899.051} C_VEL
LIN {X 0,Y 424.22,Z 580.65,A -85,B 0,C 180,E1 -9900,E2 -9900} C_VEL
LIN {X 0,Y 424.255,Z 579.626,A -85,B 0,C 180,E1 -9901.899,E2 -9901.899} C_VEL
LIN {X 0,Y 424.335,Z 578.52,A -85,B 0,C 180,E1 -9902.848,E2 -9902.848} C_VEL
LIN {X 0,Y 424.399,Z 576.973,A -85,B 0,C 180,E1 -9903.798,E2 -9903.798} C_VEL
LIN {X 0,Y 424.427,Z 573.839,A -85,B 0,C 180,E1 -9905.226,E2 -9905.226} C_VEL
LIN {X 0,Y 424.771,Z 568.71,A -85,B 0,C 180,E1 -9906.914,E2 -9906.914} C_VEL
LIN {X 0,Y 425.053,Z 562.148,A -85,B 0,C 180,E1 -9908.558,E2 -9908.558} C_VEL
LIN {X 0,Y 425.471,Z 554.853,A -85,B 0,C 180,E1 -9909.988,E2 -9909.988} C_VEL
LIN {X 0,Y 426.029,Z 545.815,A -85,B 0,C 180,E1 -9911.418,E2 -9911.418} C_VEL
LIN {X 0,Y 426.64,Z 536.552,A -85,B 0,C 180,E1 -9912.608,E2 -9912.608} C_VEL
LIN {X 0,Y 427.298,Z 526.039,A -85,B 0,C 180,E1 -9913.701,E2 -9913.701} C_VEL
LIN {X 0,Y 427.829,Z 515.058,A -85,B 0,C 180,E1 -9914.63,E2 -9914.63} C_VEL
LIN {X 0,Y 428.463,Z 502.827,A -85,B 0,C 180,E1 -9915.443,E2 -9915.443} C_VEL
LIN {X 0,Y 428.486,Z 495.488,A -85,B 0,C 180,E1 -9915.84,E2 -9915.84} C_VEL
LIN {X 0,Y 425.65,Z 482.652,A -85,B 0,C 180,E1 -9916.48,E2 -9916.48} C_VEL
LIN {X 0,Y 424.348,Z 476.844,A -85,B 0,C 180,E1 -9916.724,E2 -9916.724} C_VEL
LIN {X 0,Y 424.371,Z 474.035,A -85,B 0,C 180,E1 -9919.343,E2 -9919.343} C_VEL
LIN {X 0,Y 424.386,Z 470.839,A -85,B 0,C 180,E1 -9922.389,E2 -9922.389} C_VEL
LIN {X 0,Y 424.493,Z 467.62,A -85,B 0,C 180,E1 -9925.497,E2 -9925.497} C_VEL
LIN {X 0,Y 424.558,Z 464.385,A -85,B 0,C 180,E1 -9928.69,E2 -9928.69} C_VEL
LIN {X 0,Y 424.589,Z 463.605,A -85,B 0,C 180,E1 -9929.774,E2 -9929.774} C_VEL
LIN {X 0,Y 424.949,Z 463.553,A -85,B 0,C 180,E1 -9933.078,E2 -9933.078} C_VEL
LIN {X 0,Y 425.221,Z 463.518,A -85,B 0,C 180,E1 -9935.917,E2 -9935.917} C_VEL
LIN {X 0,Y 425.284,Z 463.508,A -85,B 0,C 180,E1 -9939.041,E2 -9939.041} C_VEL
LIN {X 0,Y 425.296,Z 463.509,A -85,B 0,C 180,E1 -9941.959,E2 -9941.959} C_VEL
LIN {X 0,Y 425.29,Z 463.508,A -85,B 0,C 180,E1 -9945.283,E2 -9945.283} C_VEL
LIN {X 0,Y 425.279,Z 463.513,A -85,B 0,C 180,E1 -9948.622,E2 -9948.622} C_VEL
LIN {X 0,Y 425.32,Z 463.504,A -85,B 0,C 180,E1 -9951.103,E2 -9951.103} C_VEL
LIN {X 0,Y 425.304,Z 463.506,A -85,B 0,C 180,E1 -9954.664,E2 -9954.664} C_VEL
LIN {X 0,Y 425.27,Z 463.513,A -85,B 0,C 180,E1 -9958.073,E2 -9958.073} C_VEL
LIN {X 0,Y 425.336,Z 463.503,A -85,B 0,C 180,E1 -9961.368,E2 -9961.368} C_VEL
LIN {X 0,Y 425.296,Z 463.509,A -85,B 0,C 180,E1 -9964.555,E2 -9964.555} C_VEL
LIN {X 0,Y 425.293,Z 463.508,A -85,B 0,C 180,E1 -9967.661,E2 -9967.661} C_VEL
LIN {X 0,Y 425.366,Z 463.5,A -85,B 0,C 180,E1 -9970.704,E2 -9970.704} C_VEL
LIN {X 0,Y 425.393,Z 463.497,A -85,B 0,C 180,E1 -9973.688,E2 -9973.688} C_VEL
LIN {X 0,Y 425.418,Z 463.492,A -85,B 0,C 180,E1 -9977.598,E2 -9977.598} C_VEL
LIN {X 0,Y 425.448,Z 463.489,A -85,B 0,C 180,E1 -9981.45,E2 -9981.45} C_VEL
LIN {X 0,Y 425.559,Z 463.476,A -85,B 0,C 180,E1 -9984.313,E2 -9984.313} C_VEL
LIN {X 0,Y 425.579,Z 463.475,A -85,B 0,C 180,E1 -9988.107,E2 -9988.107} C_VEL
LIN {X 0,Y 425.707,Z 463.459,A -85,B 0,C 180,E1 -9990,E2 -9990} C_VEL
LIN {X 0,Y 425.551,Z 463.475,A -85,B 0,C 180,E1 -9992.84,E2 -9992.84} C_VEL
LIN {X 0,Y 425.432,Z 463.49,A -85,B 0,C 180,E1 -9995.147,E2 -9995.147} C_VEL
LIN {X 0,Y 424.86,Z 463.564,A -85,B 0,C 180,E1 -9995.938,E2 -9995.938} C_VEL
LIN {X 0,Y 422,Z 463.919,A -85,B 0,C 180,E1 -9997.222,E2 -9997.222} C_VEL
LIN {X 0,Y 419.513,Z 464.23,A -85,B 0,C 180,E1 -9998.259,E2 -9998.259} C_VEL
LIN {X 0,Y 418.434,Z 464.362,A -85,B 0,C 180,E1 -9999.061,E2 -9999.061} C_VEL
LIN {X 0,Y 418.344,Z 464.373,A -85,B 0,C 180,E1 -9999.333,E2 -9999.333} C_VEL
LIN {X 0,Y 418.352,Z 464.371,A -85,B 0,C 180,E1 -10003.001,E2 -10003.001} C_VEL
LIN {X 0,Y 418.318,Z 464.376,A -85,B 0,C 180,E1 -10006.735,E2 -10006.735} C_VEL
LIN {X 0,Y 418.276,Z 464.384,A -85,B 0,C 180,E1 -10009.79,E2 -10009.79} C_VEL
LIN {X 0,Y 418.237,Z 464.387,A -85,B 0,C 180,E1 -10012.736,E2 -10012.736} C_VEL
LIN {X 0,Y 418.273,Z 464.386,A -85,B 0,C 180,E1 -10015.904,E2 -10015.904} C_VEL
LIN {X 0,Y 418.27,Z 464.383,A -85,B 0,C 180,E1 -10019.162,E2 -10019.162} C_VEL
LIN {X 0,Y 418.262,Z 464.384,A -85,B 0,C 180,E1 -10022.844,E2 -10022.844} C_VEL
LIN {X 0,Y 418.253,Z 464.386,A -85,B 0,C 180,E1 -10026.238,E2 -10026.238} C_VEL
LIN {X 0,Y 418.26,Z 464.388,A -85,B 0,C 180,E1 -10029.681,E2 -10029.681} C_VEL
LIN {X 0,Y 418.234,Z 464.388,A -85,B 0,C 180,E1 -10032.321,E2 -10032.321} C_VEL
LIN {X 0,Y 418.243,Z 464.387,A -85,B 0,C 180,E1 -10035.109,E2 -10035.109} C_VEL
LIN {X 0,Y 418.247,Z 464.388,A -85,B 0,C 180,E1 -10037.767,E2 -10037.767} C_VEL
LIN {X 0,Y 418.256,Z 464.382,A -85,B 0,C 180,E1 -10040.619,E2 -10040.619} C_VEL
LIN {X 0,Y 418.224,Z 464.389,A -85,B 0,C 180,E1 -10043.973,E2 -10043.973} C_VEL
LIN {X 0,Y 417.989,Z 464.421,A -85,B 0,C 180,E1 -10047.449,E2 -10047.449} C_VEL
LIN {X 0,Y 417.503,Z 464.483,A -85,B 0,C 180,E1 -10051.085,E2 -10051.085} C_VEL
LIN {X 0,Y 417.387,Z 464.5,A -85,B 0,C 180,E1 -10051.87,E2 -10051.87} C_VEL
LIN {X 0,Y 417.341,Z 466.575,A -85,B 0,C 180,E1 -10054.033,E2 -10054.033} C_VEL
LIN {X 0,Y 417.258,Z 470.132,A -85,B 0,C 180,E1 -10057.207,E2 -10057.207} C_VEL
LIN {X 0,Y 417.254,Z 473.957,A -85,B 0,C 180,E1 -10060.603,E2 -10060.603} C_VEL
LIN {X 0,Y 417.257,Z 477.069,A -85,B 0,C 180,E1 -10063.177,E2 -10063.177} C_VEL
LIN {X 0,Y 420.157,Z 490.305,A -85,B 0,C 180,E1 -10063.761,E2 -10063.761} C_VEL
LIN {X 0,Y 421.633,Z 497.36,A -85,B 0,C 180,E1 -10064.156,E2 -10064.156} C_VEL
LIN {X 0,Y 421.128,Z 509.567,A -85,B 0,C 180,E1 -10064.885,E2 -10064.885} C_VEL
LIN {X 0,Y 420.593,Z 520.706,A -85,B 0,C 180,E1 -10065.735,E2 -10065.735} C_VEL
LIN {X 0,Y 419.968,Z 531.972,A -85,B 0,C 180,E1 -10066.82,E2 -10066.82} C_VEL
LIN {X 0,Y 419.291,Z 541.225,A -85,B 0,C 180,E1 -10067.905,E2 -10067.905} C_VEL
LIN {X 0,Y 418.772,Z 549.756,A -85,B 0,C 180,E1 -10069.117,E2 -10069.117} C_VEL
LIN {X 0,Y 418.249,Z 558.058,A -85,B 0,C 180,E1 -10070.57,E2 -10070.57} C_VEL
LIN {X 0,Y 417.815,Z 564.759,A -85,B 0,C 180,E1 -10072.023,E2 -10072.023} C_VEL
LIN {X 0,Y 417.596,Z 570.886,A -85,B 0,C 180,E1 -10073.719,E2 -10073.719} C_VEL
LIN {X 0,Y 417.311,Z 574.859,A -85,B 0,C 180,E1 -10075.169,E2 -10075.169} C_VEL
LIN {X 0,Y 417.307,Z 576.9,A -85,B 0,C 180,E1 -10076.137,E2 -10076.137} C_VEL
LIN {X 0,Y 417.262,Z 578.533,A -85,B 0,C 180,E1 -10077.103,E2 -10077.103} C_VEL
LIN {X 0,Y 417.167,Z 579.721,A -85,B 0,C 180,E1 -10078.069,E2 -10078.069} C_VEL
LIN {X 0,Y 417.117,Z 580.845,A -85,B 0,C 180,E1 -10080,E2 -10080} C_VEL
LIN {X 0,Y 417.152,Z 580.809,A -85,B 0,C 180,E1 -10080.965,E2 -10080.965} C_VEL
LIN {X 0,Y 417.229,Z 580.32,A -85,B 0,C 180,E1 -10081.93,E2 -10081.93} C_VEL
LIN {X 0,Y 417.412,Z 578.156,A -85,B 0,C 180,E1 -10083.861,E2 -10083.861} C_VEL
LIN {X 0,Y 417.442,Z 575.413,A -85,B 0,C 180,E1 -10085.313,E2 -10085.313} C_VEL
LIN {X 0,Y 417.837,Z 570.635,A -85,B 0,C 180,E1 -10087.077,E2 -10087.077} C_VEL
LIN {X 0,Y 418.23,Z 564.76,A -85,B 0,C 180,E1 -10088.698,E2 -10088.698} C_VEL
LIN {X 0,Y 418.813,Z 558.068,A -85,B 0,C 180,E1 -10090.148,E2 -10090.148} C_VEL
LIN {X 0,Y 419.436,Z 549.704,A -85,B 0,C 180,E1 -10091.599,E2 -10091.599} C_VEL
LIN {X 0,Y 420.096,Z 541.182,A -85,B 0,C 180,E1 -10092.807,E2 -10092.807} C_VEL
LIN {X 0,Y 420.853,Z 531.638,A -85,B 0,C 180,E1 -10093.925,E2 -10093.925} C_VEL
LIN {X 0,Y 421.575,Z 520.603,A -85,B 0,C 180,E1 -10094.974,E2 -10094.974} C_VEL
LIN {X 0,Y 422.357,Z 509.556,A -85,B 0,C 180,E1 -10095.812,E2 -10095.812} C_VEL
LIN {X 0,Y 422.942,Z 499.706,A -85,B 0,C 180,E1 -10096.409,E2 -10096.409} C_VEL
LIN {X 0,Y 420.407,Z 488.794,A -85,B 0,C 180,E1 -10097.1,E2 -10097.1} C_VEL
LIN {X 0,Y 417.586,Z 479.78,A -85,B 0,C 180,E1 -10097.634,E2 -10097.634} C_VEL
LIN {X 0,Y 417.582,Z 476.394,A -85,B 0,C 180,E1 -10100.697,E2 -10100.697} C_VEL
LIN {X 0,Y 417.657,Z 472.881,A -85,B 0,C 180,E1 -10103.819,E2 -10103.819} C_VEL
LIN {X 0,Y 417.72,Z 469.232,A -85,B 0,C 180,E1 -10107.018,E2 -10107.018} C_VEL
LIN {X 0,Y 417.715,Z 465.364,A -85,B 0,C 180,E1 -10110.314,E2 -10110.314} C_VEL
LIN {X 0,Y 417.733,Z 464.651,A -85,B 0,C 180,E1 -10110.903,E2 -10110.903} C_VEL
LIN {X 0,Y 418.07,Z 464.411,A -85,B 0,C 180,E1 -10113.693,E2 -10113.693} C_VEL
LIN {X 0,Y 418.232,Z 464.39,A -85,B 0,C 180,E1 -10116.235,E2 -10116.235} C_VEL
LIN {X 0,Y 418.256,Z 464.388,A -85,B 0,C 180,E1 -10119.681,E2 -10119.681} C_VEL
LIN {X 0,Y 418.234,Z 464.391,A -85,B 0,C 180,E1 -10122.322,E2 -10122.322} C_VEL
LIN {X 0,Y 418.24,Z 464.389,A -85,B 0,C 180,E1 -10125.109,E2 -10125.109} C_VEL
LIN {X 0,Y 418.312,Z 464.533,A -85,B 0,C 180,E1 -10127.667,E2 -10127.667} C_VEL
LIN {X 0,Y 419.276,Z 470.003,A -85,B 0,C 180,E1 -10130.449,E2 -10130.449} C_VEL
LIN {X 0,Y 420.258,Z 476.043,A -85,B 0,C 180,E1 -10133.389,E2 -10133.389} C_VEL
LIN {X 0,Y 420.196,Z 480.31,A -85,B 0,C 180,E1 -10135.342,E2 -10135.342} C_VEL
LIN {X 0,Y 419.559,Z 487.979,A -85,B 0,C 180,E1 -10138.716,E2 -10138.716} C_VEL
LIN {X 0,Y 418.988,Z 495.652,A -85,B 0,C 180,E1 -10141.987,E2 -10141.987} C_VEL
LIN {X 0,Y 418.444,Z 503.312,A -85,B 0,C 180,E1 -10145.172,E2 -10145.172} C_VEL
LIN {X 0,Y 418.044,Z 510.962,A -85,B 0,C 180,E1 -10148.293,E2 -10148.293} C_VEL
LIN {X 0,Y 417.706,Z 518.614,A -85,B 0,C 180,E1 -10151.356,E2 -10151.356} C_VEL
LIN {X 0,Y 417.617,Z 522.139,A -85,B 0,C 180,E1 -10152.714,E2 -10152.714} C_VEL
LIN {X 0,Y 419.521,Z 534.745,A -85,B 0,C 180,E1 -10153.304,E2 -10153.304} C_VEL
LIN {X 0,Y 420.831,Z 547.346,A -85,B 0,C 180,E1 -10154.032,E2 -10154.032} C_VEL
LIN {X 0,Y 421.004,Z 552.961,A -85,B 0,C 180,E1 -10154.391,E2 -10154.391} C_VEL
LIN {X 0,Y 420.281,Z 565.051,A -85,B 0,C 180,E1 -10155.226,E2 -10155.226} C_VEL
LIN {X 0,Y 419.602,Z 576.126,A -85,B 0,C 180,E1 -10156.192,E2 -10156.192} C_VEL
LIN {X 0,Y 418.988,Z 586.233,A -85,B 0,C 180,E1 -10157.282,E2 -10157.282} C_VEL
LIN {X 0,Y 418.339,Z 596.203,A -85,B 0,C 180,E1 -10158.615,E2 -10158.615} C_VEL
LIN {X 0,Y 417.823,Z 605.023,A -85,B 0,C 180,E1 -10160.072,E2 -10160.072} C_VEL
LIN {X 0,Y 417.472,Z 612.069,A -85,B 0,C 180,E1 -10161.529,E2 -10161.529} C_VEL
LIN {X 0,Y 417.231,Z 618.518,A -85,B 0,C 180,E1 -10163.228,E2 -10163.228} C_VEL
LIN {X 0,Y 417.166,Z 622.735,A -85,B 0,C 180,E1 -10164.683,E2 -10164.683} C_VEL
LIN {X 0,Y 417.059,Z 625.843,A -85,B 0,C 180,E1 -10166.135,E2 -10166.135} C_VEL
LIN {X 0,Y 417.156,Z 627.38,A -85,B 0,C 180,E1 -10167.103,E2 -10167.103} C_VEL
LIN {X 0,Y 417.131,Z 628.433,A -85,B 0,C 180,E1 -10168.069,E2 -10168.069} C_VEL
LIN {X 0,Y 417.118,Z 629.069,A -85,B 0,C 180,E1 -10169.035,E2 -10169.035} C_VEL
LIN {X 0,Y 417.131,Z 629.301,A -85,B 0,C 180,E1 -10170,E2 -10170} C_VEL
LIN {X 0,Y 417.107,Z 629.113,A -85,B 0,C 180,E1 -10170.965,E2 -10170.965} C_VEL
LIN {X 0,Y 417.133,Z 628.471,A -85,B 0,C 180,E1 -10171.931,E2 -10171.931} C_VEL
LIN {X 0,Y 417.147,Z 627.416,A -85,B 0,C 180,E1 -10172.897,E2 -10172.897} C_VEL
LIN {X 0,Y 417.063,Z 625.946,A -85,B 0,C 180,E1 -10173.865,E2 -10173.865} C_VEL
LIN {X 0,Y 417.148,Z 622.882,A -85,B 0,C 180,E1 -10175.317,E2 -10175.317} C_VEL
LIN {X 0,Y 417.232,Z 618.745,A -85,B 0,C 180,E1 -10176.772,E2 -10176.772} C_VEL
LIN {X 0,Y 417.488,Z 612.426,A -85,B 0,C 180,E1 -10178.47,E2 -10178.47} C_VEL
LIN {X 0,Y 417.823,Z 605.554,A -85,B 0,C 180,E1 -10179.928,E2 -10179.928} C_VEL
LIN {X 0,Y 418.389,Z 597.086,A -85,B 0,C 180,E1 -10181.383,E2 -10181.383} C_VEL
LIN {X 0,Y 418.909,Z 588.51,A -85,B 0,C 180,E1 -10182.597,E2 -10182.597} C_VEL
LIN {X 0,Y 419.73,Z 577.501,A -85,B 0,C 180,E1 -10183.866,E2 -10183.866} C_VEL
LIN {X 0,Y 420.558,Z 566.571,A -85,B 0,C 180,E1 -10184.888,E2 -10184.888} C_VEL
LIN {X 0,Y 421.372,Z 555.532,A -85,B 0,C 180,E1 -10185.726,E2 -10185.726} C_VEL
LIN {X 0,Y 421.403,Z 548.934,A -85,B 0,C 180,E1 -10186.159,E2 -10186.159} C_VEL
LIN {X 0,Y 420.177,Z 534.327,A -85,B 0,C 180,E1 -10187.002,E2 -10187.002} C_VEL
LIN {X 0,Y 418.061,Z 522.18,A -85,B 0,C 180,E1 -10187.584,E2 -10187.584} C_VEL
LIN {X 0,Y 417.577,Z 519.52,A -85,B 0,C 180,E1 -10187.698,E2 -10187.698} C_VEL
LIN {X 0,Y 417.901,Z 510.721,A -85,B 0,C 180,E1 -10191.197,E2 -10191.197} C_VEL
LIN {X 0,Y 418.319,Z 501.933,A -85,B 0,C 180,E1 -10194.874,E2 -10194.874} C_VEL
LIN {X 0,Y 418.878,Z 494.908,A -85,B 0,C 180,E1 -10198.021,E2 -10198.021} C_VEL
LIN {X 0,Y 419.693,Z 487.166,A -85,B 0,C 180,E1 -10201.835,E2 -10201.835} C_VEL
LIN {X 0,Y 420.35,Z 482.143,A -85,B 0,C 180,E1 -10204.643,E2 -10204.643} C_VEL
LIN {X 0,Y 420.549,Z 478.558,A -85,B 0,C 180,E1 -10206.986,E2 -10206.986} C_VEL
LIN {X 0,Y 420.445,Z 476.936,A -85,B 0,C 180,E1 -10208.221,E2 -10208.221} C_VEL
LIN {X 0,Y 419.905,Z 473.799,A -85,B 0,C 180,E1 -10211.134,E2 -10211.134} C_VEL
LIN {X 0,Y 419.538,Z 471.629,A -85,B 0,C 180,E1 -10213.919,E2 -10213.919} C_VEL
LIN {X 0,Y 419.321,Z 470.292,A -85,B 0,C 180,E1 -10216.593,E2 -10216.593} C_VEL
LIN {X 0,Y 419.129,Z 469.672,A -85,B 0,C 180,E1 -10219.159,E2 -10219.159} C_VEL
LIN {X 0,Y 419.046,Z 469.61,A -85,B 0,C 180,E1 -10222.023,E2 -10222.023} C_VEL
LIN {X 0,Y 419.025,Z 469.931,A -85,B 0,C 180,E1 -10224.054,E2 -10224.054} C_VEL
LIN {X 0,Y 418.78,Z 470.882,A -85,B 0,C 180,E1 -10227.046,E2 -10227.046} C_VEL
LIN {X 0,Y 418.514,Z 472.104,A -85,B 0,C 180,E1 -10229.75,E2 -10229.75} C_VEL
LIN {X 0,Y 418.221,Z 473.963,A -85,B 0,C 180,E1 -10233.017,E2 -10233.017} C_VEL
LIN {X 0,Y 418.018,Z 476.046,A -85,B 0,C 180,E1 -10236.203,E2 -10236.203} C_VEL
LIN {X 0,Y 417.802,Z 478.333,A -85,B 0,C 180,E1 -10239.314,E2 -10239.314} C_VEL
LIN {X 0,Y 417.699,Z 480.811,A -85,B 0,C 180,E1 -10242.447,E2 -10242.447} C_VEL
LIN {X 0,Y 421.698,Z 493.708,A -85,B 0,C 180,E1 -10243.24,E2 -10243.24} C_VEL
LIN {X 0,Y 422.948,Z 500.152,A -85,B 0,C 180,E1 -10243.654,E2 -10243.654} C_VEL
LIN {X 0,Y 422.278,Z 512.496,A -85,B 0,C 180,E1 -10244.433,E2 -10244.433} C_VEL
LIN {X 0,Y 421.503,Z 523.831,A -85,B 0,C 180,E1 -10245.35,E2 -10245.35} C_VEL
LIN {X 0,Y 420.645,Z 534.96,A -85,B 0,C 180,E1 -10246.473,E2 -10246.473} C_VEL
LIN {X 0,Y 419.877,Z 544.57,A -85,B 0,C 180,E1 -10247.678,E2 -10247.678} C_VEL
LIN {X 0,Y 419.11,Z 553.978,A -85,B 0,C 180,E1 -10249.126,E2 -10249.126} C_VEL
LIN {X 0,Y 418.57,Z 561.5,A -85,B 0,C 180,E1 -10250.578,E2 -10250.578} C_VEL
LIN {X 0,Y 417.98,Z 568.418,A -85,B 0,C 180,E1 -10252.27,E2 -10252.27} C_VEL
LIN {X 0,Y 417.679,Z 573,A -85,B 0,C 180,E1 -10253.721,E2 -10253.721} C_VEL
LIN {X 0,Y 417.51,Z 576.475,A -85,B 0,C 180,E1 -10255.172,E2 -10255.172} C_VEL
LIN {X 0,Y 417.415,Z 578.247,A -85,B 0,C 180,E1 -10256.139,E2 -10256.139} C_VEL
LIN {X 0,Y 417.292,Z 579.558,A -85,B 0,C 180,E1 -10257.104,E2 -10257.104} C_VEL
LIN {X 0,Y 417.256,Z 580.465,A -85,B 0,C 180,E1 -10258.07,E2 -10258.07} C_VEL
LIN {X 0,Y 417.182,Z 580.982,A -85,B 0,C 180,E1 -10259.035,E2 -10259.035} C_VEL
LIN {X 0,Y 417.133,Z 581.07,A -85,B 0,C 180,E1 -10260,E2 -10260} C_VEL
LIN {X 0,Y 417.123,Z 580.735,A -85,B 0,C 180,E1 -10260.966,E2 -10260.966} C_VEL
LIN {X 0,Y 417.178,Z 580.002,A -85,B 0,C 180,E1 -10261.931,E2 -10261.931} C_VEL
LIN {X 0,Y 417.269,Z 578.872,A -85,B 0,C 180,E1 -10262.897,E2 -10262.897} C_VEL
LIN {X 0,Y 417.301,Z 576.35,A -85,B 0,C 180,E1 -10264.347,E2 -10264.347} C_VEL
LIN {X 0,Y 417.473,Z 572.811,A -85,B 0,C 180,E1 -10265.797,E2 -10265.797} C_VEL
LIN {X 0,Y 417.716,Z 568.169,A -85,B 0,C 180,E1 -10267.249,E2 -10267.249} C_VEL
LIN {X 0,Y 418.077,Z 561.132,A -85,B 0,C 180,E1 -10268.946,E2 -10268.946} C_VEL
LIN {X 0,Y 418.55,Z 553.524,A -85,B 0,C 180,E1 -10270.4,E2 -10270.4} C_VEL
LIN {X 0,Y 419.038,Z 545.782,A -85,B 0,C 180,E1 -10271.611,E2 -10271.611} C_VEL
LIN {X 0,Y 419.798,Z 535.325,A -85,B 0,C 180,E1 -10272.939,E2 -10272.939} C_VEL
LIN {X 0,Y 420.398,Z 523.971,A -85,B 0,C 180,E1 -10274.104,E2 -10274.104} C_VEL
LIN {X 0,Y 420.979,Z 513.03,A -85,B 0,C 180,E1 -10274.997,E2 -10274.997} C_VEL
LIN {X 0,Y 421.648,Z 500.824,A -85,B 0,C 180,E1 -10275.776,E2 -10275.776} C_VEL
LIN {X 0,Y 421.449,Z 496.057,A -85,B 0,C 180,E1 -10276.041,E2 -10276.041} C_VEL
LIN {X 0,Y 418.52,Z 482.963,A -85,B 0,C 180,E1 -10276.714,E2 -10276.714} C_VEL
LIN {X 0,Y 417.265,Z 477.198,A -85,B 0,C 180,E1 -10276.953,E2 -10276.953} C_VEL
LIN {X 0,Y 417.3,Z 474.29,A -85,B 0,C 180,E1 -10279.684,E2 -10279.684} C_VEL
LIN {X 0,Y 417.318,Z 471.053,A -85,B 0,C 180,E1 -10282.789,E2 -10282.789} C_VEL
LIN {X 0,Y 417.426,Z 467.802,A -85,B 0,C 180,E1 -10285.961,E2 -10285.961} C_VEL
LIN {X 0,Y 417.5,Z 464.537,A -85,B 0,C 180,E1 -10289.221,E2 -10289.221} C_VEL
LIN {X 0,Y 417.878,Z 464.436,A -85,B 0,C 180,E1 -10292.561,E2 -10292.561} C_VEL
LIN {X 0,Y 418.119,Z 464.403,A -85,B 0,C 180,E1 -10294.855,E2 -10294.855} C_VEL
LIN {X 0,Y 418.227,Z 464.389,A -85,B 0,C 180,E1 -10297.833,E2 -10297.833} C_VEL
LIN {X 0,Y 418.226,Z 464.386,A -85,B 0,C 180,E1 -10300.948,E2 -10300.948} C_VEL
LIN {X 0,Y 418.221,Z 464.39,A -85,B 0,C 180,E1 -10303.731,E2 -10303.731} C_VEL
LIN {X 0,Y 418.213,Z 464.391,A -85,B 0,C 180,E1 -10306.449,E2 -10306.449} C_VEL
LIN {X 0,Y 418.229,Z 464.388,A -85,B 0,C 180,E1 -10309.13,E2 -10309.13} C_VEL
LIN {X 0,Y 418.238,Z 464.389,A -85,B 0,C 180,E1 -10312.166,E2 -10312.166} C_VEL
LIN {X 0,Y 418.27,Z 464.382,A -85,B 0,C 180,E1 -10315.42,E2 -10315.42} C_VEL
LIN {X 0,Y 418.216,Z 464.391,A -85,B 0,C 180,E1 -10318.604,E2 -10318.604} C_VEL
LIN {X 0,Y 418.296,Z 464.381,A -85,B 0,C 180,E1 -10321.937,E2 -10321.937} C_VEL
LIN {X 0,Y 418.295,Z 464.378,A -85,B 0,C 180,E1 -10325.163,E2 -10325.163} C_VEL
LIN {X 0,Y 418.239,Z 464.388,A -85,B 0,C 180,E1 -10328.304,E2 -10328.304} C_VEL
LIN {X 0,Y 418.286,Z 464.381,A -85,B 0,C 180,E1 -10331.383,E2 -10331.383} C_VEL
LIN {X 0,Y 418.308,Z 464.381,A -85,B 0,C 180,E1 -10334.406,E2 -10334.406} C_VEL
LIN {X 0,Y 418.361,Z 464.37,A -85,B 0,C 180,E1 -10337.386,E2 -10337.386} C_VEL
LIN {X 0,Y 418.405,Z 464.365,A -85,B 0,C 180,E1 -10341.305,E2 -10341.305} C_VEL
LIN {X 0,Y 418.518,Z 464.353,A -85,B 0,C 180,E1 -10344.217,E2 -10344.217} C_VEL
LIN {X 0,Y 418.548,Z 464.351,A -85,B 0,C 180,E1 -10348.075,E2 -10348.075} C_VEL
LIN {X 0,Y 418.677,Z 464.335,A -85,B 0,C 180,E1 -10350,E2 -10350} C_VEL
LIN {X 0,Y 418.506,Z 464.352,A -85,B 0,C 180,E1 -10352.888,E2 -10352.888} C_VEL
LIN {X 0,Y 418.504,Z 464.356,A -85,B 0,C 180,E1 -10355.783,E2 -10355.783} C_VEL
LIN {X 0,Y 418.383,Z 464.369,A -85,B 0,C 180,E1 -10358.695,E2 -10358.695} C_VEL
LIN {X 0,Y 418.344,Z 464.373,A -85,B 0,C 180,E1 -10359.333,E2 -10359.333} C_VEL
LIN {X 0,Y 417.676,Z 464.46,A -85,B 0,C 180,E1 -10360.137,E2 -10360.137} C_VEL
LIN {X 0,Y 414.833,Z 464.811,A -85,B 0,C 180,E1 -10361.442,E2 -10361.442} C_VEL
LIN {X 0,Y 412.417,Z 465.111,A -85,B 0,C 180,E1 -10362.496,E2 -10362.496} C_VEL
LIN {X 0,Y 411.365,Z 465.242,A -85,B 0,C 180,E1 -10363.311,E2 -10363.311} C_VEL
LIN {X 0,Y 411.27,Z 465.255,A -85,B 0,C 180,E1 -10363.587,E2 -10363.587} C_VEL
LIN {X 0,Y 411.262,Z 465.255,A -85,B 0,C 180,E1 -10366.889,E2 -10366.889} C_VEL
LIN {X 0,Y 411.236,Z 465.261,A -85,B 0,C 180,E1 -10369.987,E2 -10369.987} C_VEL
LIN {X 0,Y 411.201,Z 465.263,A -85,B 0,C 180,E1 -10373.148,E2 -10373.148} C_VEL
LIN {X 0,Y 411.242,Z 465.257,A -85,B 0,C 180,E1 -10376.381,E2 -10376.381} C_VEL
LIN {X 0,Y 411.205,Z 465.266,A -85,B 0,C 180,E1 -10379.712,E2 -10379.712} C_VEL
LIN {X 0,Y 411.211,Z 465.263,A -85,B 0,C 180,E1 -10383.156,E2 -10383.156} C_VEL
LIN {X 0,Y 411.2,Z 465.263,A -85,B 0,C 180,E1 -10386.553,E2 -10386.553} C_VEL
LIN {X 0,Y 411.223,Z 465.265,A -85,B 0,C 180,E1 -10389.729,E2 -10389.729} C_VEL
LIN {X 0,Y 411.178,Z 465.267,A -85,B 0,C 180,E1 -10393.133,E2 -10393.133} C_VEL
LIN {X 0,Y 411.177,Z 465.268,A -85,B 0,C 180,E1 -10395.88,E2 -10395.88} C_VEL
LIN {X 0,Y 411.168,Z 465.266,A -85,B 0,C 180,E1 -10398.771,E2 -10398.771} C_VEL
LIN {X 0,Y 411.207,Z 465.265,A -85,B 0,C 180,E1 -10401.831,E2 -10401.831} C_VEL
LIN {X 0,Y 411.113,Z 465.275,A -85,B 0,C 180,E1 -10405.142,E2 -10405.142} C_VEL
LIN {X 0,Y 410.832,Z 465.313,A -85,B 0,C 180,E1 -10407.973,E2 -10407.973} C_VEL
LIN {X 0,Y 410.409,Z 465.367,A -85,B 0,C 180,E1 -10411.348,E2 -10411.348} C_VEL
LIN {X 0,Y 410.298,Z 465.435,A -85,B 0,C 180,E1 -10412.452,E2 -10412.452} C_VEL
LIN {X 0,Y 410.234,Z 469.092,A -85,B 0,C 180,E1 -10415.722,E2 -10415.722} C_VEL
LIN {X 0,Y 410.183,Z 472.658,A -85,B 0,C 180,E1 -10418.911,E2 -10418.911} C_VEL
LIN {X 0,Y 410.146,Z 476.167,A -85,B 0,C 180,E1 -10422.035,E2 -10422.035} C_VEL
LIN {X 0,Y 410.158,Z 477.168,A -85,B 0,C 180,E1 -10422.904,E2 -10422.904} C_VEL
LIN {X 0,Y 413.564,Z 492.954,A -85,B 0,C 180,E1 -10423.662,E2 -10423.662} C_VEL
LIN {X 0,Y 414.741,Z 499.09,A -85,B 0,C 180,E1 -10424.021,E2 -10424.021} C_VEL
LIN {X 0,Y 414.147,Z 510.851,A -85,B 0,C 180,E1 -10424.75,E2 -10424.75} C_VEL
LIN {X 0,Y 413.564,Z 522.629,A -85,B 0,C 180,E1 -10425.695,E2 -10425.695} C_VEL
LIN {X 0,Y 412.88,Z 534.032,A -85,B 0,C 180,E1 -10426.84,E2 -10426.84} C_VEL
LIN {X 0,Y 412.2,Z 542.993,A -85,B 0,C 180,E1 -10427.944,E2 -10427.944} C_VEL
LIN {X 0,Y 411.55,Z 552.727,A -85,B 0,C 180,E1 -10429.422,E2 -10429.422} C_VEL
LIN {X 0,Y 411.047,Z 560.579,A -85,B 0,C 180,E1 -10430.9,E2 -10430.9} C_VEL
LIN {X 0,Y 410.646,Z 567.764,A -85,B 0,C 180,E1 -10432.625,E2 -10432.625} C_VEL
LIN {X 0,Y 410.415,Z 572.562,A -85,B 0,C 180,E1 -10434.102,E2 -10434.102} C_VEL
LIN {X 0,Y 410.214,Z 576.229,A -85,B 0,C 180,E1 -10435.578,E2 -10435.578} C_VEL
LIN {X 0,Y 410.198,Z 578.857,A -85,B 0,C 180,E1 -10437.053,E2 -10437.053} C_VEL
LIN {X 0,Y 410.095,Z 580.085,A -85,B 0,C 180,E1 -10438.036,E2 -10438.036} C_VEL
LIN {X 0,Y 410.034,Z 581.251,A -85,B 0,C 180,E1 -10440,E2 -10440} C_VEL
LIN {X 0,Y 410.071,Z 581.244,A -85,B 0,C 180,E1 -10440.982,E2 -10440.982} C_VEL
LIN {X 0,Y 410.153,Z 580.787,A -85,B 0,C 180,E1 -10441.964,E2 -10441.964} C_VEL
LIN {X 0,Y 410.363,Z 578.672,A -85,B 0,C 180,E1 -10443.928,E2 -10443.928} C_VEL
LIN {X 0,Y 410.386,Z 575.972,A -85,B 0,C 180,E1 -10445.404,E2 -10445.404} C_VEL
LIN {X 0,Y 410.818,Z 571.411,A -85,B 0,C 180,E1 -10447.147,E2 -10447.147} C_VEL
LIN {X 0,Y 411.24,Z 565.412,A -85,B 0,C 180,E1 -10448.847,E2 -10448.847} C_VEL
LIN {X 0,Y 411.872,Z 558.772,A -85,B 0,C 180,E1 -10450.321,E2 -10450.321} C_VEL
LIN {X 0,Y 412.541,Z 550.528,A -85,B 0,C 180,E1 -10451.796,E2 -10451.796} C_VEL
LIN {X 0,Y 413.249,Z 542.138,A -85,B 0,C 180,E1 -10453.023,E2 -10453.023} C_VEL
LIN {X 0,Y 414.058,Z 532.737,A -85,B 0,C 180,E1 -10454.156,E2 -10454.156} C_VEL
LIN {X 0,Y 414.837,Z 521.847,A -85,B 0,C 180,E1 -10455.223,E2 -10455.223} C_VEL
LIN {X 0,Y 415.77,Z 509.271,A -85,B 0,C 180,E1 -10456.195,E2 -10456.195} C_VEL
LIN {X 0,Y 416.164,Z 500.258,A -85,B 0,C 180,E1 -10456.759,E2 -10456.759} C_VEL
LIN {X 0,Y 413.547,Z 489.612,A -85,B 0,C 180,E1 -10457.481,E2 -10457.481} C_VEL
LIN {X 0,Y 410.562,Z 480.337,A -85,B 0,C 180,E1 -10458.043,E2 -10458.043} C_VEL
LIN {X 0,Y 410.566,Z 477.017,A -85,B 0,C 180,E1 -10461.068,E2 -10461.068} C_VEL
LIN {X 0,Y 410.644,Z 473.488,A -85,B 0,C 180,E1 -10464.252,E2 -10464.252} C_VEL
LIN {X 0,Y 410.683,Z 469.776,A -85,B 0,C 180,E1 -10467.519,E2 -10467.519} C_VEL
LIN {X 0,Y 410.745,Z 465.964,A -85,B 0,C 180,E1 -10470.885,E2 -10470.885} C_VEL
LIN {X 0,Y 410.83,Z 465.314,A -85,B 0,C 180,E1 -10472.026,E2 -10472.026} C_VEL
LIN {X 0,Y 411.113,Z 465.278,A -85,B 0,C 180,E1 -10474.858,E2 -10474.858} C_VEL
LIN {X 0,Y 411.208,Z 465.266,A -85,B 0,C 180,E1 -10478.169,E2 -10478.169} C_VEL
LIN {X 0,Y 411.167,Z 465.27,A -85,B 0,C 180,E1 -10481.229,E2 -10481.229} C_VEL
LIN {X 0,Y 411.182,Z 465.267,A -85,B 0,C 180,E1 -10484.49,E2 -10484.49} C_VEL
LIN {X 0,Y 411.286,Z 465.464,A -85,B 0,C 180,E1 -10487.44,E2 -10487.44} C_VEL
LIN {X 0,Y 412.469,Z 472.198,A -85,B 0,C 180,E1 -10490.917,E2 -10490.917} C_VEL
LIN {X 0,Y 413.277,Z 477.39,A -85,B 0,C 180,E1 -10493.473,E2 -10493.473} C_VEL
LIN {X 0,Y 413.179,Z 481.275,A -85,B 0,C 180,E1 -10495.278,E2 -10495.278} C_VEL
LIN {X 0,Y 412.548,Z 488.251,A -85,B 0,C 180,E1 -10498.406,E2 -10498.406} C_VEL
LIN {X 0,Y 412.02,Z 495.275,A -85,B 0,C 180,E1 -10501.471,E2 -10501.471} C_VEL
LIN {X 0,Y 411.425,Z 503.272,A -85,B 0,C 180,E1 -10504.871,E2 -10504.871} C_VEL
LIN {X 0,Y 410.935,Z 511.818,A -85,B 0,C 180,E1 -10508.426,E2 -10508.426} C_VEL
LIN {X 0,Y 410.615,Z 519.438,A -85,B 0,C 180,E1 -10511.54,E2 -10511.54} C_VEL
LIN {X 0,Y 410.542,Z 521.276,A -85,B 0,C 180,E1 -10512.286,E2 -10512.286} C_VEL
LIN {X 0,Y 412.411,Z 532.473,A -85,B 0,C 180,E1 -10512.829,E2 -10512.829} C_VEL
LIN {X 0,Y 413.723,Z 544.695,A -85,B 0,C 180,E1 -10513.536,E2 -10513.536} C_VEL
LIN {X 0,Y 414.308,Z 551.753,A -85,B 0,C 180,E1 -10514.021,E2 -10514.021} C_VEL
LIN {X 0,Y 413.376,Z 564.534,A -85,B 0,C 180,E1 -10514.973,E2 -10514.973} C_VEL
LIN {X 0,Y 412.503,Z 577.622,A -85,B 0,C 180,E1 -10516.2,E2 -10516.2} C_VEL
LIN {X 0,Y 411.791,Z 588.313,A -85,B 0,C 180,E1 -10517.432,E2 -10517.432} C_VEL
LIN {X 0,Y 411.237,Z 597.067,A -85,B 0,C 180,E1 -10518.666,E2 -10518.666} C_VEL
LIN {X 0,Y 410.712,Z 605.605,A -85,B 0,C 180,E1 -10520.147,E2 -10520.147} C_VEL
LIN {X 0,Y 410.36,Z 612.461,A -85,B 0,C 180,E1 -10521.629,E2 -10521.629} C_VEL
LIN {X 0,Y 410.163,Z 617.937,A -85,B 0,C 180,E1 -10523.111,E2 -10523.111} C_VEL
LIN {X 0,Y 410.08,Z 622.193,A -85,B 0,C 180,E1 -10524.591,E2 -10524.591} C_VEL
LIN {X 0,Y 409.976,Z 625.337,A -85,B 0,C 180,E1 -10526.068,E2 -10526.068} C_VEL
LIN {X 0,Y 410.07,Z 626.893,A -85,B 0,C 180,E1 -10527.053,E2 -10527.053} C_VEL
LIN {X 0,Y 410.058,Z 627.975,A -85,B 0,C 180,E1 -10528.036,E2 -10528.036} C_VEL
LIN {X 0,Y 410.037,Z 628.624,A -85,B 0,C 180,E1 -10529.018,E2 -10529.018} C_VEL
LIN {X 0,Y 410.047,Z 628.868,A -85,B 0,C 180,E1 -10530,E2 -10530} C_VEL
LIN {X 0,Y 410.026,Z 628.7,A -85,B 0,C 180,E1 -10530.982,E2 -10530.982} C_VEL
LIN {X 0,Y 410.059,Z 628.077,A -85,B 0,C 180,E1 -10531.964,E2 -10531.964} C_VEL
LIN {X 0,Y 410.045,Z 627.032,A -85,B 0,C 180,E1 -10532.947,E2 -10532.947} C_VEL
LIN {X 0,Y 409.979,Z 625.57,A -85,B 0,C 180,E1 -10533.932,E2 -10533.932} C_VEL
LIN {X 0,Y 410.042,Z 622.528,A -85,B 0,C 180,E1 -10535.409,E2 -10535.409} C_VEL
LIN {X 0,Y 410.164,Z 618.421,A -85,B 0,C 180,E1 -10536.889,E2 -10536.889} C_VEL
LIN {X 0,Y 410.444,Z 612.154,A -85,B 0,C 180,E1 -10538.617,E2 -10538.617} C_VEL
LIN {X 0,Y 410.83,Z 604.044,A -85,B 0,C 180,E1 -10540.348,E2 -10540.348} C_VEL
LIN {X 0,Y 411.506,Z 595.342,A -85,B 0,C 180,E1 -10541.826,E2 -10541.826} C_VEL
LIN {X 0,Y 412.242,Z 584.88,A -85,B 0,C 180,E1 -10543.262,E2 -10543.262} C_VEL
LIN {X 0,Y 413.044,Z 574.994,A -85,B 0,C 180,E1 -10544.372,E2 -10544.372} C_VEL
LIN {X 0,Y 413.95,Z 563.909,A -85,B 0,C 180,E1 -10545.384,E2 -10545.384} C_VEL
LIN {X 0,Y 414.75,Z 552.387,A -85,B 0,C 180,E1 -10546.236,E2 -10546.236} C_VEL
LIN {X 0,Y 413.894,Z 539.483,A -85,B 0,C 180,E1 -10547.068,E2 -10547.068} C_VEL
LIN {X 0,Y 412.161,Z 526.917,A -85,B 0,C 180,E1 -10547.743,E2 -10547.743} C_VEL
LIN {X 0,Y 410.508,Z 518.922,A -85,B 0,C 180,E1 -10548.142,E2 -10548.142} C_VEL
LIN {X 0,Y 410.885,Z 510.509,A -85,B 0,C 180,E1 -10551.577,E2 -10551.577} C_VEL
LIN {X 0,Y 411.362,Z 501.924,A -85,B 0,C 180,E1 -10555.285,E2 -10555.285} C_VEL
LIN {X 0,Y 411.911,Z 494.917,A -85,B 0,C 180,E1 -10558.538,E2 -10558.538} C_VEL
LIN {X 0,Y 412.707,Z 488.375,A -85,B 0,C 180,E1 -10561.864,E2 -10561.864} C_VEL
LIN {X 0,Y 413.241,Z 484.363,A -85,B 0,C 180,E1 -10564.141,E2 -10564.141} C_VEL
LIN {X 0,Y 413.601,Z 480.707,A -85,B 0,C 180,E1 -10566.493,E2 -10566.493} C_VEL
LIN {X 0,Y 413.341,Z 477.537,A -85,B 0,C 180,E1 -10568.985,E2 -10568.985} C_VEL
LIN {X 0,Y 412.897,Z 474.939,A -85,B 0,C 180,E1 -10571.593,E2 -10571.593} C_VEL
LIN {X 0,Y 412.565,Z 472.951,A -85,B 0,C 180,E1 -10574.319,E2 -10574.319} C_VEL
LIN {X 0,Y 412.336,Z 471.651,A -85,B 0,C 180,E1 -10577.131,E2 -10577.131} C_VEL
LIN {X 0,Y 412.147,Z 471.064,A -85,B 0,C 180,E1 -10580.117,E2 -10580.117} C_VEL
LIN {X 0,Y 412.089,Z 471.198,A -85,B 0,C 180,E1 -10583.351,E2 -10583.351} C_VEL
LIN {X 0,Y 411.907,Z 471.748,A -85,B 0,C 180,E1 -10585.733,E2 -10585.733} C_VEL
LIN {X 0,Y 411.594,Z 473.076,A -85,B 0,C 180,E1 -10589.186,E2 -10589.186} C_VEL
LIN {X 0,Y 411.225,Z 474.94,A -85,B 0,C 180,E1 -10592.711,E2 -10592.711} C_VEL
LIN {X 0,Y 411.016,Z 476.852,A -85,B 0,C 180,E1 -10595.772,E2 -10595.772} C_VEL
LIN {X 0,Y 410.796,Z 479.083,A -85,B 0,C 180,E1 -10598.945,E2 -10598.945} C_VEL
LIN {X 0,Y 410.676,Z 481.366,A -85,B 0,C 180,E1 -10601.93,E2 -10601.93} C_VEL
LIN {X 0,Y 410.686,Z 481.442,A -85,B 0,C 180,E1 -10602.027,E2 -10602.027} C_VEL
LIN {X 0,Y 414.674,Z 493.732,A -85,B 0,C 180,E1 -10602.821,E2 -10602.821} C_VEL
LIN {X 0,Y 416.289,Z 500.968,A -85,B 0,C 180,E1 -10603.322,E2 -10603.322} C_VEL
LIN {X 0,Y 415.565,Z 513.925,A -85,B 0,C 180,E1 -10604.175,E2 -10604.175} C_VEL
LIN {X 0,Y 414.715,Z 525.407,A -85,B 0,C 180,E1 -10605.136,E2 -10605.136} C_VEL
LIN {X 0,Y 413.827,Z 536.039,A -85,B 0,C 180,E1 -10606.246,E2 -10606.246} C_VEL
LIN {X 0,Y 413.002,Z 545.517,A -85,B 0,C 180,E1 -10607.469,E2 -10607.469} C_VEL
LIN {X 0,Y 412.185,Z 554.785,A -85,B 0,C 180,E1 -10608.941,E2 -10608.941} C_VEL
LIN {X 0,Y 411.616,Z 562.199,A -85,B 0,C 180,E1 -10610.417,E2 -10610.417} C_VEL
LIN {X 0,Y 410.989,Z 569.077,A -85,B 0,C 180,E1 -10612.137,E2 -10612.137} C_VEL
LIN {X 0,Y 410.653,Z 573.621,A -85,B 0,C 180,E1 -10613.613,E2 -10613.613} C_VEL
LIN {X 0,Y 410.457,Z 577.055,A -85,B 0,C 180,E1 -10615.089,E2 -10615.089} C_VEL
LIN {X 0,Y 410.367,Z 578.784,A -85,B 0,C 180,E1 -10616.072,E2 -10616.072} C_VEL
LIN {X 0,Y 410.177,Z 580.949,A -85,B 0,C 180,E1 -10618.036,E2 -10618.036} C_VEL
LIN {X 0,Y 410.099,Z 581.44,A -85,B 0,C 180,E1 -10619.018,E2 -10619.018} C_VEL
LIN {X 0,Y 410.048,Z 581.491,A -85,B 0,C 180,E1 -10620,E2 -10620} C_VEL
LIN {X 0,Y 410.105,Z 580.377,A -85,B 0,C 180,E1 -10621.964,E2 -10621.964} C_VEL
LIN {X 0,Y 410.204,Z 579.217,A -85,B 0,C 180,E1 -10622.946,E2 -10622.946} C_VEL
LIN {X 0,Y 410.217,Z 576.654,A -85,B 0,C 180,E1 -10624.422,E2 -10624.422} C_VEL
LIN {X 0,Y 410.415,Z 573.064,A -85,B 0,C 180,E1 -10625.898,E2 -10625.898} C_VEL
LIN {X 0,Y 410.673,Z 568.359,A -85,B 0,C 180,E1 -10627.374,E2 -10627.374} C_VEL
LIN {X 0,Y 411.044,Z 561.242,A -85,B 0,C 180,E1 -10629.1,E2 -10629.1} C_VEL
LIN {X 0,Y 411.535,Z 553.565,A -85,B 0,C 180,E1 -10630.579,E2 -10630.579} C_VEL
LIN {X 0,Y 412.05,Z 545.74,A -85,B 0,C 180,E1 -10631.811,E2 -10631.811} C_VEL
LIN {X 0,Y 412.866,Z 535.163,A -85,B 0,C 180,E1 -10633.161,E2 -10633.161} C_VEL
LIN {X 0,Y 413.487,Z 523.691,A -85,B 0,C 180,E1 -10634.344,E2 -10634.344} C_VEL
LIN {X 0,Y 414.1,Z 512.559,A -85,B 0,C 180,E1 -10635.252,E2 -10635.252} C_VEL
LIN {X 0,Y 414.789,Z 499.262,A -85,B 0,C 180,E1 -10636.098,E2 -10636.098} C_VEL
LIN {X 0,Y 412.292,Z 486.848,A -85,B 0,C 180,E1 -10636.781,E2 -10636.781} C_VEL
LIN {X 0,Y 410.179,Z 477.539,A -85,B 0,C 180,E1 -10637.199,E2 -10637.199} C_VEL
LIN {X 0,Y 410.212,Z 474.54,A -85,B 0,C 180,E1 -10640.039,E2 -10640.039} C_VEL
LIN {X 0,Y 410.261,Z 471.258,A -85,B 0,C 180,E1 -10643.204,E2 -10643.204} C_VEL
LIN {X 0,Y 410.376,Z 467.977,A -85,B 0,C 180,E1 -10646.441,E2 -10646.441} C_VEL
LIN {X 0,Y 410.439,Z 465.368,A -85,B 0,C 180,E1 -10649.158,E2 -10649.158} C_VEL
LIN {X 0,Y 410.748,Z 465.324,A -85,B 0,C 180,E1 -10652.034,E2 -10652.034} C_VEL
LIN {X 0,Y 411.081,Z 465.28,A -85,B 0,C 180,E1 -10654.852,E2 -10654.852} C_VEL
LIN {X 0,Y 411.203,Z 465.265,A -85,B 0,C 180,E1 -10658.168,E2 -10658.168} C_VEL
LIN {X 0,Y 411.168,Z 465.265,A -85,B 0,C 180,E1 -10661.229,E2 -10661.229} C_VEL
LIN {X 0,Y 411.184,Z 465.266,A -85,B 0,C 180,E1 -10664.49,E2 -10664.49} C_VEL
LIN {X 0,Y 411.182,Z 465.267,A -85,B 0,C 180,E1 -10668.195,E2 -10668.195} C_VEL
LIN {X 0,Y 411.228,Z 465.26,A -85,B 0,C 180,E1 -10670.777,E2 -10670.777} C_VEL
LIN {X 0,Y 411.203,Z 465.264,A -85,B 0,C 180,E1 -10674.472,E2 -10674.472} C_VEL
LIN {X 0,Y 411.212,Z 465.262,A -85,B 0,C 180,E1 -10676.874,E2 -10676.874} C_VEL
LIN {X 0,Y 411.238,Z 465.261,A -85,B 0,C 180,E1 -10680.644,E2 -10680.644} C_VEL
LIN {X 0,Y 411.242,Z 465.258,A -85,B 0,C 180,E1 -10683.619,E2 -10683.619} C_VEL
LIN {X 0,Y 411.207,Z 465.261,A -85,B 0,C 180,E1 -10686.853,E2 -10686.853} C_VEL
LIN {X 0,Y 411.22,Z 465.263,A -85,B 0,C 180,E1 -10690.05,E2 -10690.05} C_VEL
LIN {X 0,Y 411.268,Z 465.255,A -85,B 0,C 180,E1 -10693.131,E2 -10693.131} C_VEL
LIN {X 0,Y 411.311,Z 465.248,A -85,B 0,C 180,E1 -10696.896,E2 -10696.896} C_VEL
LIN {X 0,Y 411.297,Z 465.253,A -85,B 0,C 180,E1 -10700.161,E2 -10700.161} C_VEL
LIN {X 0,Y 411.487,Z 465.229,A -85,B 0,C 180,E1 -10702.147,E2 -10702.147} C_VEL
LIN {X 0,Y 411.48,Z 465.23,A -85,B 0,C 180,E1 -10704.118,E2 -10704.118} C_VEL
LIN {X 0,Y 411.517,Z 465.226,A -85,B 0,C 180,E1 -10708.043,E2 -10708.043} C_VEL
LIN {X 0,Y 411.646,Z 465.211,A -85,B 0,C 180,E1 -10710,E2 -10710} C_VEL
LIN {X 0,Y 411.463,Z 465.229,A -85,B 0,C 180,E1 -10712.937,E2 -10712.937} C_VEL
LIN {X 0,Y 411.429,Z 465.235,A -85,B 0,C 180,E1 -10716.868,E2 -10716.868} C_VEL
LIN {X 0,Y 411.297,Z 465.253,A -85,B 0,C 180,E1 -10719.839,E2 -10719.839} C_VEL
LIN {X 0,Y 411.311,Z 465.248,A -85,B 0,C 180,E1 -10723.104,E2 -10723.104} C_VEL
LIN {X 0,Y 411.27,Z 465.255,A -85,B 0,C 180,E1 -10723.587,E2 -10723.587} C_VEL
LIN {X 0,Y 410.574,Z 465.346,A -85,B 0,C 180,E1 -10724.405,E2 -10724.405} C_VEL
LIN {X 0,Y 407.695,Z 465.703,A -85,B 0,C 180,E1 -10725.733,E2 -10725.733} C_VEL
LIN {X 0,Y 405.287,Z 465.999,A -85,B 0,C 180,E1 -10726.806,E2 -10726.806} C_VEL
LIN {X 0,Y 404.272,Z 466.13,A -85,B 0,C 180,E1 -10727.635,E2 -10727.635} C_VEL
LIN {X 0,Y 404.199,Z 466.135,A -85,B 0,C 180,E1 -10727.916,E2 -10727.916} C_VEL
LIN {X 0,Y 404.169,Z 466.141,A -85,B 0,C 180,E1 -10730.351,E2 -10730.351} C_VEL
LIN {X 0,Y 404.168,Z 466.14,A -85,B 0,C 180,E1 -10733.575,E2 -10733.575} C_VEL
LIN {X 0,Y 404.188,Z 466.14,A -85,B 0,C 180,E1 -10735.766,E2 -10735.766} C_VEL
LIN {X 0,Y 404.2,Z 466.137,A -85,B 0,C 180,E1 -10737.999,E2 -10737.999} C_VEL
LIN {X 0,Y 404.144,Z 466.145,A -85,B 0,C 180,E1 -10741.558,E2 -10741.558} C_VEL
LIN {X 0,Y 404.19,Z 466.136,A -85,B 0,C 180,E1 -10745.016,E2 -10745.016} C_VEL
LIN {X 0,Y 404.164,Z 466.137,A -85,B 0,C 180,E1 -10748.756,E2 -10748.756} C_VEL
LIN {X 0,Y 404.128,Z 466.148,A -85,B 0,C 180,E1 -10751.6,E2 -10751.6} C_VEL
LIN {X 0,Y 404.151,Z 466.142,A -85,B 0,C 180,E1 -10754.522,E2 -10754.522} C_VEL
LIN {X 0,Y 404.144,Z 466.144,A -85,B 0,C 180,E1 -10757.296,E2 -10757.296} C_VEL
LIN {X 0,Y 404.173,Z 466.141,A -85,B 0,C 180,E1 -10759.955,E2 -10759.955} C_VEL
LIN {X 0,Y 404.132,Z 466.143,A -85,B 0,C 180,E1 -10763.126,E2 -10763.126} C_VEL
LIN {X 0,Y 403.973,Z 466.166,A -85,B 0,C 180,E1 -10766.171,E2 -10766.171} C_VEL
LIN {X 0,Y 403.696,Z 466.199,A -85,B 0,C 180,E1 -10768.545,E2 -10768.545} C_VEL
LIN {X 0,Y 403.287,Z 466.256,A -85,B 0,C 180,E1 -10771.931,E2 -10771.931} C_VEL
LIN {X 0,Y 403.225,Z 466.374,A -85,B 0,C 180,E1 -10772.736,E2 -10772.736} C_VEL
LIN {X 0,Y 403.124,Z 470.417,A -85,B 0,C 180,E1 -10776.36,E2 -10776.36} C_VEL
LIN {X 0,Y 403.091,Z 474.042,A -85,B 0,C 180,E1 -10779.591,E2 -10779.591} C_VEL
LIN {X 0,Y 403.092,Z 477.594,A -85,B 0,C 180,E1 -10782.693,E2 -10782.693} C_VEL
LIN {X 0,Y 405.898,Z 490.526,A -85,B 0,C 180,E1 -10783.28,E2 -10783.28} C_VEL
LIN {X 0,Y 407.812,Z 500.308,A -85,B 0,C 180,E1 -10783.852,E2 -10783.852} C_VEL
LIN {X 0,Y 407.168,Z 512.069,A -85,B 0,C 180,E1 -10784.61,E2 -10784.61} C_VEL
LIN {X 0,Y 406.553,Z 524.602,A -85,B 0,C 180,E1 -10785.66,E2 -10785.66} C_VEL
LIN {X 0,Y 405.869,Z 534.916,A -85,B 0,C 180,E1 -10786.736,E2 -10786.736} C_VEL
LIN {X 0,Y 405.092,Z 544.646,A -85,B 0,C 180,E1 -10787.983,E2 -10787.983} C_VEL
LIN {X 0,Y 404.463,Z 554.173,A -85,B 0,C 180,E1 -10789.487,E2 -10789.487} C_VEL
LIN {X 0,Y 403.957,Z 561.776,A -85,B 0,C 180,E1 -10790.991,E2 -10790.991} C_VEL
LIN {X 0,Y 403.605,Z 567.901,A -85,B 0,C 180,E1 -10792.496,E2 -10792.496} C_VEL
LIN {X 0,Y 403.355,Z 572.757,A -85,B 0,C 180,E1 -10793.999,E2 -10793.999} C_VEL
LIN {X 0,Y 403.133,Z 576.479,A -85,B 0,C 180,E1 -10795.5,E2 -10795.5} C_VEL
LIN {X 0,Y 403.134,Z 579.159,A -85,B 0,C 180,E1 -10797.002,E2 -10797.002} C_VEL
LIN {X 0,Y 403.025,Z 580.433,A -85,B 0,C 180,E1 -10798.001,E2 -10798.001} C_VEL
LIN {X 0,Y 402.953,Z 581.245,A -85,B 0,C 180,E1 -10799,E2 -10799} C_VEL
LIN {X 0,Y 402.992,Z 581.679,A -85,B 0,C 180,E1 -10800.999,E2 -10800.999} C_VEL
LIN {X 0,Y 403.079,Z 581.265,A -85,B 0,C 180,E1 -10801.998,E2 -10801.998} C_VEL
LIN {X 0,Y 403.315,Z 579.191,A -85,B 0,C 180,E1 -10803.997,E2 -10803.997} C_VEL
LIN {X 0,Y 403.334,Z 576.532,A -85,B 0,C 180,E1 -10805.499,E2 -10805.499} C_VEL
LIN {X 0,Y 403.803,Z 572.184,A -85,B 0,C 180,E1 -10807.224,E2 -10807.224} C_VEL
LIN {X 0,Y 404.266,Z 566.121,A -85,B 0,C 180,E1 -10809.001,E2 -10809.001} C_VEL
LIN {X 0,Y 404.937,Z 559.576,A -85,B 0,C 180,E1 -10810.5,E2 -10810.5} C_VEL
LIN {X 0,Y 405.479,Z 552.927,A -85,B 0,C 180,E1 -10811.751,E2 -10811.751} C_VEL
LIN {X 0,Y 406.132,Z 544.948,A -85,B 0,C 180,E1 -10813,E2 -10813} C_VEL
LIN {X 0,Y 407.114,Z 535.551,A -85,B 0,C 180,E1 -10814.196,E2 -10814.196} C_VEL
LIN {X 0,Y 408.031,Z 524.426,A -85,B 0,C 180,E1 -10815.368,E2 -10815.368} C_VEL
LIN {X 0,Y 408.96,Z 512.687,A -85,B 0,C 180,E1 -10816.344,E2 -10816.344} C_VEL
LIN {X 0,Y 409.606,Z 501.935,A -85,B 0,C 180,E1 -10817.058,E2 -10817.058} C_VEL
LIN {X 0,Y 406.948,Z 491.21,A -85,B 0,C 180,E1 -10817.821,E2 -10817.821} C_VEL
LIN {X 0,Y 403.553,Z 480.867,A -85,B 0,C 180,E1 -10818.532,E2 -10818.532} C_VEL
LIN {X 0,Y 403.56,Z 477.712,A -85,B 0,C 180,E1 -10821.451,E2 -10821.451} C_VEL
LIN {X 0,Y 403.691,Z 473.669,A -85,B 0,C 180,E1 -10825.137,E2 -10825.137} C_VEL
LIN {X 0,Y 403.696,Z 470.457,A -85,B 0,C 180,E1 -10828.037,E2 -10828.037} C_VEL
LIN {X 0,Y 403.771,Z 466.578,A -85,B 0,C 180,E1 -10831.478,E2 -10831.478} C_VEL
LIN {X 0,Y 403.94,Z 466.171,A -85,B 0,C 180,E1 -10833.37,E2 -10833.37} C_VEL
LIN {X 0,Y 404.121,Z 466.148,A -85,B 0,C 180,E1 -10836.248,E2 -10836.248} C_VEL
LIN {X 0,Y 404.159,Z 466.142,A -85,B 0,C 180,E1 -10838.756,E2 -10838.756} C_VEL
LIN {X 0,Y 404.127,Z 466.146,A -85,B 0,C 180,E1 -10841.6,E2 -10841.6} C_VEL
LIN {X 0,Y 404.151,Z 466.143,A -85,B 0,C 180,E1 -10844.523,E2 -10844.523} C_VEL
LIN {X 0,Y 404.19,Z 466.202,A -85,B 0,C 180,E1 -10847.107,E2 -10847.107} C_VEL
LIN {X 0,Y 405.192,Z 471.804,A -85,B 0,C 180,E1 -10850.077,E2 -10850.077} C_VEL
LIN {X 0,Y 406.086,Z 477.088,A -85,B 0,C 180,E1 -10852.76,E2 -10852.76} C_VEL
LIN {X 0,Y 406.311,Z 480.449,A -85,B 0,C 180,E1 -10854.387,E2 -10854.387} C_VEL
LIN {X 0,Y 405.71,Z 487.246,A -85,B 0,C 180,E1 -10857.52,E2 -10857.52} C_VEL
LIN {X 0,Y 405.067,Z 494.886,A -85,B 0,C 180,E1 -10860.935,E2 -10860.935} C_VEL
LIN {X 0,Y 404.394,Z 503.432,A -85,B 0,C 180,E1 -10864.651,E2 -10864.651} C_VEL
LIN {X 0,Y 403.918,Z 511.381,A -85,B 0,C 180,E1 -10868.032,E2 -10868.032} C_VEL
LIN {X 0,Y 403.514,Z 520.391,A -85,B 0,C 180,E1 -10871.795,E2 -10871.795} C_VEL
LIN {X 0,Y 405.698,Z 532.822,A -85,B 0,C 180,E1 -10872.47,E2 -10872.47} C_VEL
LIN {X 0,Y 406.972,Z 545.67,A -85,B 0,C 180,E1 -10873.255,E2 -10873.255} C_VEL
LIN {X 0,Y 407.529,Z 552.545,A -85,B 0,C 180,E1 -10873.748,E2 -10873.748} C_VEL
LIN {X 0,Y 406.533,Z 564.97,A -85,B 0,C 180,E1 -10874.714,E2 -10874.714} C_VEL
LIN {X 0,Y 405.586,Z 577.469,A -85,B 0,C 180,E1 -10875.96,E2 -10875.96} C_VEL
LIN {X 0,Y 404.82,Z 587.545,A -85,B 0,C 180,E1 -10877.212,E2 -10877.212} C_VEL
LIN {X 0,Y 404.114,Z 597.823,A -85,B 0,C 180,E1 -10878.717,E2 -10878.717} C_VEL
LIN {X 0,Y 403.587,Z 606.115,A -85,B 0,C 180,E1 -10880.225,E2 -10880.225} C_VEL
LIN {X 0,Y 403.256,Z 612.809,A -85,B 0,C 180,E1 -10881.733,E2 -10881.733} C_VEL
LIN {X 0,Y 403.057,Z 618.491,A -85,B 0,C 180,E1 -10883.353,E2 -10883.353} C_VEL
LIN {X 0,Y 403.018,Z 622.819,A -85,B 0,C 180,E1 -10884.998,E2 -10884.998} C_VEL
LIN {X 0,Y 402.896,Z 624.813,A -85,B 0,C 180,E1 -10885.999,E2 -10885.999} C_VEL
LIN {X 0,Y 402.971,Z 626.388,A -85,B 0,C 180,E1 -10887.001,E2 -10887.001} C_VEL
LIN {X 0,Y 402.987,Z 627.509,A -85,B 0,C 180,E1 -10888.001,E2 -10888.001} C_VEL
LIN {X 0,Y 402.959,Z 628.174,A -85,B 0,C 180,E1 -10889.001,E2 -10889.001} C_VEL
LIN {X 0,Y 402.965,Z 628.432,A -85,B 0,C 180,E1 -10890,E2 -10890} C_VEL
LIN {X 0,Y 402.949,Z 628.282,A -85,B 0,C 180,E1 -10890.999,E2 -10890.999} C_VEL
LIN {X 0,Y 402.987,Z 627.687,A -85,B 0,C 180,E1 -10891.999,E2 -10891.999} C_VEL
LIN {X 0,Y 402.943,Z 626.654,A -85,B 0,C 180,E1 -10892.999,E2 -10892.999} C_VEL
LIN {X 0,Y 402.897,Z 625.206,A -85,B 0,C 180,E1 -10894.001,E2 -10894.001} C_VEL
LIN {X 0,Y 402.941,Z 622.189,A -85,B 0,C 180,E1 -10895.505,E2 -10895.505} C_VEL
LIN {X 0,Y 403.076,Z 618.118,A -85,B 0,C 180,E1 -10897.011,E2 -10897.011} C_VEL
LIN {X 0,Y 403.376,Z 611.915,A -85,B 0,C 180,E1 -10898.769,E2 -10898.769} C_VEL
LIN {X 0,Y 403.76,Z 605.127,A -85,B 0,C 180,E1 -10900.278,E2 -10900.278} C_VEL
LIN {X 0,Y 404.417,Z 596.792,A -85,B 0,C 180,E1 -10901.782,E2 -10901.782} C_VEL
LIN {X 0,Y 405.126,Z 586.867,A -85,B 0,C 180,E1 -10903.242,E2 -10903.242} C_VEL
LIN {X 0,Y 406.11,Z 575.953,A -85,B 0,C 180,E1 -10904.533,E2 -10904.533} C_VEL
LIN {X 0,Y 407.144,Z 564.32,A -85,B 0,C 180,E1 -10905.647,E2 -10905.647} C_VEL
LIN {X 0,Y 407.955,Z 553.082,A -85,B 0,C 180,E1 -10906.514,E2 -10906.514} C_VEL
LIN {X 0,Y 407.063,Z 538.701,A -85,B 0,C 180,E1 -10907.477,E2 -10907.477} C_VEL
LIN {X 0,Y 405.239,Z 526.583,A -85,B 0,C 180,E1 -10908.166,E2 -10908.166} C_VEL
LIN {X 0,Y 403.48,Z 518.343,A -85,B 0,C 180,E1 -10908.601,E2 -10908.601} C_VEL
LIN {X 0,Y 403.859,Z 510.337,A -85,B 0,C 180,E1 -10911.972,E2 -10911.972} C_VEL
LIN {X 0,Y 404.414,Z 501.848,A -85,B 0,C 180,E1 -10915.751,E2 -10915.751} C_VEL
LIN {X 0,Y 405.032,Z 494.958,A -85,B 0,C 180,E1 -10919.068,E2 -10919.068} C_VEL
LIN {X 0,Y 405.833,Z 488.572,A -85,B 0,C 180,E1 -10922.469,E2 -10922.469} C_VEL
LIN {X 0,Y 406.395,Z 484.677,A -85,B 0,C 180,E1 -10924.798,E2 -10924.798} C_VEL
LIN {X 0,Y 406.629,Z 481.021,A -85,B 0,C 180,E1 -10927.34,E2 -10927.34} C_VEL
LIN {X 0,Y 406.246,Z 478.175,A -85,B 0,C 180,E1 -10929.799,E2 -10929.799} C_VEL
LIN {X 0,Y 405.846,Z 475.767,A -85,B 0,C 180,E1 -10932.482,E2 -10932.482} C_VEL
LIN {X 0,Y 405.522,Z 473.983,A -85,B 0,C 180,E1 -10935.281,E2 -10935.281} C_VEL
LIN {X 0,Y 405.329,Z 472.878,A -85,B 0,C 180,E1 -10938.209,E2 -10938.209} C_VEL
LIN {X 0,Y 405.159,Z 472.502,A -85,B 0,C 180,E1 -10941.357,E2 -10941.357} C_VEL
LIN {X 0,Y 405.081,Z 472.695,A -85,B 0,C 180,E1 -10943.851,E2 -10943.851} C_VEL
LIN {X 0,Y 404.861,Z 473.312,A -85,B 0,C 180,E1 -10946.433,E2 -10946.433} C_VEL
LIN {X 0,Y 404.675,Z 474.1,A -85,B 0,C 180,E1 -10948.6,E2 -10948.6} C_VEL
LIN {X 0,Y 404.278,Z 475.734,A -85,B 0,C 180,E1 -10952.007,E2 -10952.007} C_VEL
LIN {X 0,Y 404.028,Z 477.682,A -85,B 0,C 180,E1 -10955.325,E2 -10955.325} C_VEL
LIN {X 0,Y 403.787,Z 479.852,A -85,B 0,C 180,E1 -10958.561,E2 -10958.561} C_VEL
LIN {X 0,Y 403.69,Z 482.099,A -85,B 0,C 180,E1 -10961.574,E2 -10961.574} C_VEL
LIN {X 0,Y 408.085,Z 495.368,A -85,B 0,C 180,E1 -10962.49,E2 -10962.49} C_VEL
LIN {X 0,Y 409.634,Z 501.868,A -85,B 0,C 180,E1 -10962.964,E2 -10962.964} C_VEL
LIN {X 0,Y 408.978,Z 514.007,A -85,B 0,C 180,E1 -10963.785,E2 -10963.785} C_VEL
LIN {X 0,Y 408.079,Z 525.521,A -85,B 0,C 180,E1 -10964.769,E2 -10964.769} C_VEL
LIN {X 0,Y 407.129,Z 536.109,A -85,B 0,C 180,E1 -10965.89,E2 -10965.89} C_VEL
LIN {X 0,Y 406.137,Z 546.494,A -85,B 0,C 180,E1 -10967.254,E2 -10967.254} C_VEL
LIN {X 0,Y 405.274,Z 555.668,A -85,B 0,C 180,E1 -10968.75,E2 -10968.75} C_VEL
LIN {X 0,Y 404.668,Z 562.987,A -85,B 0,C 180,E1 -10970.251,E2 -10970.251} C_VEL
LIN {X 0,Y 404.011,Z 569.765,A -85,B 0,C 180,E1 -10972.001,E2 -10972.001} C_VEL
LIN {X 0,Y 403.628,Z 574.241,A -85,B 0,C 180,E1 -10973.502,E2 -10973.502} C_VEL
LIN {X 0,Y 403.407,Z 577.636,A -85,B 0,C 180,E1 -10975.003,E2 -10975.003} C_VEL
LIN {X 0,Y 403.321,Z 579.322,A -85,B 0,C 180,E1 -10976.003,E2 -10976.003} C_VEL
LIN {X 0,Y 403.171,Z 580.584,A -85,B 0,C 180,E1 -10977.003,E2 -10977.003} C_VEL
LIN {X 0,Y 403.101,Z 581.443,A -85,B 0,C 180,E1 -10978.002,E2 -10978.002} C_VEL
LIN {X 0,Y 403.019,Z 581.901,A -85,B 0,C 180,E1 -10979.001,E2 -10979.001} C_VEL
LIN {X 0,Y 402.967,Z 581.914,A -85,B 0,C 180,E1 -10980,E2 -10980} C_VEL
LIN {X 0,Y 402.964,Z 581.528,A -85,B 0,C 180,E1 -10981,E2 -10981} C_VEL
LIN {X 0,Y 403.035,Z 580.743,A -85,B 0,C 180,E1 -10981.999,E2 -10981.999} C_VEL
LIN {X 0,Y 403.14,Z 579.537,A -85,B 0,C 180,E1 -10982.998,E2 -10982.998} C_VEL
LIN {X 0,Y 403.137,Z 576.926,A -85,B 0,C 180,E1 -10984.5,E2 -10984.5} C_VEL
LIN {X 0,Y 403.357,Z 573.28,A -85,B 0,C 180,E1 -10986.001,E2 -10986.001} C_VEL
LIN {X 0,Y 403.619,Z 568.506,A -85,B 0,C 180,E1 -10987.504,E2 -10987.504} C_VEL
LIN {X 0,Y 404.034,Z 561.323,A -85,B 0,C 180,E1 -10989.259,E2 -10989.259} C_VEL
LIN {X 0,Y 404.542,Z 553.568,A -85,B 0,C 180,E1 -10990.764,E2 -10990.764} C_VEL
LIN {X 0,Y 405.204,Z 543.857,A -85,B 0,C 180,E1 -10992.267,E2 -10992.267} C_VEL
LIN {X 0,Y 405.999,Z 533.913,A -85,B 0,C 180,E1 -10993.515,E2 -10993.515} C_VEL
LIN {X 0,Y 406.597,Z 523.244,A -85,B 0,C 180,E1 -10994.601,E2 -10994.601} C_VEL
LIN {X 0,Y 407.222,Z 512.094,A -85,B 0,C 180,E1 -10995.516,E2 -10995.516} C_VEL
LIN {X 0,Y 407.794,Z 499.436,A -85,B 0,C 180,E1 -10996.332,E2 -10996.332} C_VEL
LIN {X 0,Y 405.119,Z 487.017,A -85,B 0,C 180,E1 -10997.028,E2 -10997.028} C_VEL
LIN {X 0,Y 403.133,Z 477.889,A -85,B 0,C 180,E1 -10997.436,E2 -10997.436} C_VEL
LIN {X 0,Y 403.153,Z 474.777,A -85,B 0,C 180,E1 -11000.405,E2 -11000.405} C_VEL
LIN {X 0,Y 403.183,Z 471.466,A -85,B 0,C 180,E1 -11003.636,E2 -11003.636} C_VEL
LIN {X 0,Y 403.339,Z 468.144,A -85,B 0,C 180,E1 -11006.939,E2 -11006.939} C_VEL
LIN {X 0,Y 403.404,Z 466.243,A -85,B 0,C 180,E1 -11009.197,E2 -11009.197} C_VEL
LIN {X 0,Y 403.772,Z 466.192,A -85,B 0,C 180,E1 -11012.656,E2 -11012.656} C_VEL
LIN {X 0,Y 404.047,Z 466.154,A -85,B 0,C 180,E1 -11015.162,E2 -11015.162} C_VEL
LIN {X 0,Y 404.152,Z 466.144,A -85,B 0,C 180,E1 -11018.507,E2 -11018.507} C_VEL
LIN {X 0,Y 404.128,Z 466.143,A -85,B 0,C 180,E1 -11021.6,E2 -11021.6} C_VEL
LIN {X 0,Y 404.153,Z 466.142,A -85,B 0,C 180,E1 -11024.523,E2 -11024.523} C_VEL
LIN {X 0,Y 404.14,Z 466.143,A -85,B 0,C 180,E1 -11027.296,E2 -11027.296} C_VEL
LIN {X 0,Y 404.173,Z 466.14,A -85,B 0,C 180,E1 -11029.956,E2 -11029.956} C_VEL
LIN {X 0,Y 404.143,Z 466.14,A -85,B 0,C 180,E1 -11033.125,E2 -11033.125} C_VEL
LIN {X 0,Y 404.149,Z 466.144,A -85,B 0,C 180,E1 -11036.188,E2 -11036.188} C_VEL
LIN {X 0,Y 404.15,Z 466.144,A -85,B 0,C 180,E1 -11039.715,E2 -11039.715} C_VEL
LIN {X 0,Y 404.199,Z 466.135,A -85,B 0,C 180,E1 -11043.123,E2 -11043.123} C_VEL
LIN {X 0,Y 404.181,Z 466.136,A -85,B 0,C 180,E1 -11045.335,E2 -11045.335} C_VEL
LIN {X 0,Y 404.144,Z 466.143,A -85,B 0,C 180,E1 -11048.581,E2 -11048.581} C_VEL
LIN {X 0,Y 404.214,Z 466.137,A -85,B 0,C 180,E1 -11051.762,E2 -11051.762} C_VEL
LIN {X 0,Y 404.212,Z 466.134,A -85,B 0,C 180,E1 -11054.882,E2 -11054.882} C_VEL
LIN {X 0,Y 404.261,Z 466.13,A -85,B 0,C 180,E1 -11057.959,E2 -11057.959} C_VEL
LIN {X 0,Y 404.439,Z 466.108,A -85,B 0,C 180,E1 -11062.1,E2 -11062.1} C_VEL
LIN {X 0,Y 404.429,Z 466.109,A -85,B 0,C 180,E1 -11064.015,E2 -11064.015} C_VEL
LIN {X 0,Y 404.486,Z 466.102,A -85,B 0,C 180,E1 -11068.009,E2 -11068.009} C_VEL
LIN {X 0,Y 404.615,Z 466.087,A -85,B 0,C 180,E1 -11070,E2 -11070} C_VEL
LIN {X 0,Y 404.421,Z 466.106,A -85,B 0,C 180,E1 -11072.988,E2 -11072.988} C_VEL
LIN {X 0,Y 404.375,Z 466.113,A -85,B 0,C 180,E1 -11076.988,E2 -11076.988} C_VEL
LIN {X 0,Y 404.262,Z 466.13,A -85,B 0,C 180,E1 -11080.012,E2 -11080.012} C_VEL
LIN {X 0,Y 404.272,Z 466.125,A -85,B 0,C 180,E1 -11083.211,E2 -11083.211} C_VEL
LIN {X 0,Y 404.221,Z 466.132,A -85,B 0,C 180,E1 -11087.007,E2 -11087.007} C_VEL
LIN {X 0,Y 404.199,Z 466.135,A -85,B 0,C 180,E1 -11087.916,E2 -11087.916} C_VEL
LIN {X 0,Y 403.548,Z 466.219,A -85,B 0,C 180,E1 -11088.748,E2 -11088.748} C_VEL
LIN {X 0,Y 400.667,Z 466.579,A -85,B 0,C 180,E1 -11090.099,E2 -11090.099} C_VEL
LIN {X 0,Y 398.217,Z 466.883,A -85,B 0,C 180,E1 -11091.191,E2 -11091.191} C_VEL
LIN {X 0,Y 397.169,Z 467.014,A -85,B 0,C 180,E1 -11092.036,E2 -11092.036} C_VEL
LIN {X 0,Y 397.086,Z 467.02,A -85,B 0,C 180,E1 -11092.322,E2 -11092.322} C_VEL
LIN {X 0,Y 397.157,Z 467.013,A -85,B 0,C 180,E1 -11095.512,E2 -11095.512} C_VEL
LIN {X 0,Y 397.127,Z 467.016,A -85,B 0,C 180,E1 -11098.543,E2 -11098.543} C_VEL
LIN {X 0,Y 397.083,Z 467.024,A -85,B 0,C 180,E1 -11102.071,E2 -11102.071} C_VEL
LIN {X 0,Y 397.125,Z 467.018,A -85,B 0,C 180,E1 -11105.503,E2 -11105.503} C_VEL
LIN {X 0,Y 397.138,Z 467.013,A -85,B 0,C 180,E1 -11108.862,E2 -11108.862} C_VEL
LIN {X 0,Y 397.073,Z 467.024,A -85,B 0,C 180,E1 -11112.267,E2 -11112.267} C_VEL
LIN {X 0,Y 397.094,Z 467.021,A -85,B 0,C 180,E1 -11115.068,E2 -11115.068} C_VEL
LIN {X 0,Y 397.072,Z 467.026,A -85,B 0,C 180,E1 -11118.02,E2 -11118.02} C_VEL
LIN {X 0,Y 397.133,Z 467.015,A -85,B 0,C 180,E1 -11121.138,E2 -11121.138} C_VEL
LIN {X 0,Y 397.03,Z 467.028,A -85,B 0,C 180,E1 -11124.515,E2 -11124.515} C_VEL
LIN {X 0,Y 396.886,Z 467.046,A -85,B 0,C 180,E1 -11126.705,E2 -11126.705} C_VEL
LIN {X 0,Y 396.445,Z 467.104,A -85,B 0,C 180,E1 -11130.302,E2 -11130.302} C_VEL
LIN {X 0,Y 396.187,Z 467.139,A -85,B 0,C 180,E1 -11132.534,E2 -11132.534} C_VEL
LIN {X 0,Y 396.101,Z 469.302,A -85,B 0,C 180,E1 -11134.809,E2 -11134.809} C_VEL
LIN {X 0,Y 396.045,Z 472.997,A -85,B 0,C 180,E1 -11138.12,E2 -11138.12} C_VEL
LIN {X 0,Y 395.993,Z 476.633,A -85,B 0,C 180,E1 -11141.369,E2 -11141.369} C_VEL
LIN {X 0,Y 396.032,Z 478.013,A -85,B 0,C 180,E1 -11142.457,E2 -11142.457} C_VEL
LIN {X 0,Y 398.933,Z 491.485,A -85,B 0,C 180,E1 -11143.09,E2 -11143.09} C_VEL
LIN {X 0,Y 400.824,Z 500.703,A -85,B 0,C 180,E1 -11143.648,E2 -11143.648} C_VEL
LIN {X 0,Y 400.181,Z 512.998,A -85,B 0,C 180,E1 -11144.465,E2 -11144.465} C_VEL
LIN {X 0,Y 399.559,Z 525.078,A -85,B 0,C 180,E1 -11145.501,E2 -11145.501} C_VEL
LIN {X 0,Y 398.843,Z 535.633,A -85,B 0,C 180,E1 -11146.628,E2 -11146.628} C_VEL
LIN {X 0,Y 398.016,Z 546.189,A -85,B 0,C 180,E1 -11148.025,E2 -11148.025} C_VEL
LIN {X 0,Y 397.445,Z 554.069,A -85,B 0,C 180,E1 -11149.299,E2 -11149.299} C_VEL
LIN {X 0,Y 396.919,Z 561.795,A -85,B 0,C 180,E1 -11150.83,E2 -11150.83} C_VEL
LIN {X 0,Y 396.541,Z 567.998,A -85,B 0,C 180,E1 -11152.361,E2 -11152.361} C_VEL
LIN {X 0,Y 396.298,Z 572.927,A -85,B 0,C 180,E1 -11153.892,E2 -11153.892} C_VEL
LIN {X 0,Y 396.058,Z 576.717,A -85,B 0,C 180,E1 -11155.42,E2 -11155.42} C_VEL
LIN {X 0,Y 396.053,Z 579.458,A -85,B 0,C 180,E1 -11156.948,E2 -11156.948} C_VEL
LIN {X 0,Y 395.957,Z 580.769,A -85,B 0,C 180,E1 -11157.965,E2 -11157.965} C_VEL
LIN {X 0,Y 395.879,Z 581.625,A -85,B 0,C 180,E1 -11158.983,E2 -11158.983} C_VEL
LIN {X 0,Y 395.875,Z 582.066,A -85,B 0,C 180,E1 -11160,E2 -11160} C_VEL
LIN {X 0,Y 395.916,Z 582.112,A -85,B 0,C 180,E1 -11161.017,E2 -11161.017} C_VEL
LIN {X 0,Y 396.008,Z 581.741,A -85,B 0,C 180,E1 -11162.034,E2 -11162.034} C_VEL
LIN {X 0,Y 396.268,Z 579.722,A -85,B 0,C 180,E1 -11164.068,E2 -11164.068} C_VEL
LIN {X 0,Y 396.287,Z 577.129,A -85,B 0,C 180,E1 -11165.597,E2 -11165.597} C_VEL
LIN {X 0,Y 396.776,Z 573.042,A -85,B 0,C 180,E1 -11167.289,E2 -11167.289} C_VEL
LIN {X 0,Y 397.148,Z 568.733,A -85,B 0,C 180,E1 -11168.651,E2 -11168.651} C_VEL
LIN {X 0,Y 397.769,Z 562.719,A -85,B 0,C 180,E1 -11170.177,E2 -11170.177} C_VEL
LIN {X 0,Y 398.446,Z 555.201,A -85,B 0,C 180,E1 -11171.703,E2 -11171.703} C_VEL
LIN {X 0,Y 399.293,Z 545.988,A -85,B 0,C 180,E1 -11173.227,E2 -11173.227} C_VEL
LIN {X 0,Y 400.346,Z 536.724,A -85,B 0,C 180,E1 -11174.451,E2 -11174.451} C_VEL
LIN {X 0,Y 401.404,Z 524.694,A -85,B 0,C 180,E1 -11175.746,E2 -11175.746} C_VEL
LIN {X 0,Y 402.436,Z 512.725,A -85,B 0,C 180,E1 -11176.747,E2 -11176.747} C_VEL
LIN {X 0,Y 403.06,Z 503.997,A -85,B 0,C 180,E1 -11177.343,E2 -11177.343} C_VEL
LIN {X 0,Y 400.995,Z 494.866,A -85,B 0,C 180,E1 -11178.045,E2 -11178.045} C_VEL
LIN {X 0,Y 397.246,Z 483.772,A -85,B 0,C 180,E1 -11178.843,E2 -11178.843} C_VEL
LIN {X 0,Y 396.562,Z 481.451,A -85,B 0,C 180,E1 -11179.005,E2 -11179.005} C_VEL
LIN {X 0,Y 396.605,Z 477.237,A -85,B 0,C 180,E1 -11182.945,E2 -11182.945} C_VEL
LIN {X 0,Y 396.696,Z 473.633,A -85,B 0,C 180,E1 -11186.289,E2 -11186.289} C_VEL
LIN {X 0,Y 396.759,Z 469.846,A -85,B 0,C 180,E1 -11189.777,E2 -11189.777} C_VEL
LIN {X 0,Y 396.773,Z 467.311,A -85,B 0,C 180,E1 -11192.099,E2 -11192.099} C_VEL
LIN {X 0,Y 396.97,Z 467.039,A -85,B 0,C 180,E1 -11194.509,E2 -11194.509} C_VEL
LIN {X 0,Y 397.093,Z 467.024,A -85,B 0,C 180,E1 -11197.208,E2 -11197.208} C_VEL
LIN {X 0,Y 397.104,Z 467.02,A -85,B 0,C 180,E1 -11200.446,E2 -11200.446} C_VEL
LIN {X 0,Y 397.105,Z 467.022,A -85,B 0,C 180,E1 -11203.648,E2 -11203.648} C_VEL
LIN {X 0,Y 397.157,Z 467.046,A -85,B 0,C 180,E1 -11206.839,E2 -11206.839} C_VEL
LIN {X 0,Y 398.19,Z 472.887,A -85,B 0,C 180,E1 -11209.992,E2 -11209.992} C_VEL
LIN {X 0,Y 399.212,Z 479.188,A -85,B 0,C 180,E1 -11213.233,E2 -11213.233} C_VEL
LIN {X 0,Y 399.157,Z 483.03,A -85,B 0,C 180,E1 -11215.094,E2 -11215.094} C_VEL
LIN {X 0,Y 398.419,Z 490.667,A -85,B 0,C 180,E1 -11218.643,E2 -11218.643} C_VEL
LIN {X 0,Y 397.814,Z 498.196,A -85,B 0,C 180,E1 -11222.047,E2 -11222.047} C_VEL
LIN {X 0,Y 397.217,Z 505.876,A -85,B 0,C 180,E1 -11225.431,E2 -11225.431} C_VEL
LIN {X 0,Y 396.751,Z 513.453,A -85,B 0,C 180,E1 -11228.707,E2 -11228.707} C_VEL
LIN {X 0,Y 396.47,Z 519.593,A -85,B 0,C 180,E1 -11231.326,E2 -11231.326} C_VEL
LIN {X 0,Y 399.047,Z 533.482,A -85,B 0,C 180,E1 -11232.103,E2 -11232.103} C_VEL
LIN {X 0,Y 400.246,Z 546.432,A -85,B 0,C 180,E1 -11232.941,E2 -11232.941} C_VEL
LIN {X 0,Y 400.646,Z 554.852,A -85,B 0,C 180,E1 -11233.577,E2 -11233.577} C_VEL
LIN {X 0,Y 399.632,Z 566.777,A -85,B 0,C 180,E1 -11234.574,E2 -11234.574} C_VEL
LIN {X 0,Y 398.696,Z 577.736,A -85,B 0,C 180,E1 -11235.713,E2 -11235.713} C_VEL
LIN {X 0,Y 397.891,Z 587.639,A -85,B 0,C 180,E1 -11236.985,E2 -11236.985} C_VEL
LIN {X 0,Y 397.105,Z 597.372,A -85,B 0,C 180,E1 -11238.515,E2 -11238.515} C_VEL
LIN {X 0,Y 396.412,Z 607.796,A -85,B 0,C 180,E1 -11240.561,E2 -11240.561} C_VEL
LIN {X 0,Y 396.057,Z 614.964,A -85,B 0,C 180,E1 -11242.352,E2 -11242.352} C_VEL
LIN {X 0,Y 395.909,Z 619.72,A -85,B 0,C 180,E1 -11243.886,E2 -11243.886} C_VEL
LIN {X 0,Y 395.878,Z 623.324,A -85,B 0,C 180,E1 -11245.418,E2 -11245.418} C_VEL
LIN {X 0,Y 395.875,Z 625.867,A -85,B 0,C 180,E1 -11246.947,E2 -11246.947} C_VEL
LIN {X 0,Y 395.917,Z 627.029,A -85,B 0,C 180,E1 -11247.965,E2 -11247.965} C_VEL
LIN {X 0,Y 395.883,Z 627.716,A -85,B 0,C 180,E1 -11248.983,E2 -11248.983} C_VEL
LIN {X 0,Y 395.886,Z 627.993,A -85,B 0,C 180,E1 -11250,E2 -11250} C_VEL
LIN {X 0,Y 395.874,Z 627.859,A -85,B 0,C 180,E1 -11251.017,E2 -11251.017} C_VEL
LIN {X 0,Y 395.915,Z 627.301,A -85,B 0,C 180,E1 -11252.035,E2 -11252.035} C_VEL
LIN {X 0,Y 395.843,Z 626.282,A -85,B 0,C 180,E1 -11253.053,E2 -11253.053} C_VEL
LIN {X 0,Y 395.817,Z 624.853,A -85,B 0,C 180,E1 -11254.073,E2 -11254.073} C_VEL
LIN {X 0,Y 395.84,Z 621.372,A -85,B 0,C 180,E1 -11255.825,E2 -11255.825} C_VEL
LIN {X 0,Y 396.061,Z 616.25,A -85,B 0,C 180,E1 -11257.648,E2 -11257.648} C_VEL
LIN {X 0,Y 396.429,Z 609.599,A -85,B 0,C 180,E1 -11259.438,E2 -11259.438} C_VEL
LIN {X 0,Y 396.905,Z 602.434,A -85,B 0,C 180,E1 -11260.973,E2 -11260.973} C_VEL
LIN {X 0,Y 397.679,Z 593.586,A -85,B 0,C 180,E1 -11262.503,E2 -11262.503} C_VEL
LIN {X 0,Y 398.528,Z 583.544,A -85,B 0,C 180,E1 -11263.919,E2 -11263.919} C_VEL
LIN {X 0,Y 399.578,Z 572.657,A -85,B 0,C 180,E1 -11265.167,E2 -11265.167} C_VEL
LIN {X 0,Y 400.763,Z 560.355,A -85,B 0,C 180,E1 -11266.295,E2 -11266.295} C_VEL
LIN {X 0,Y 401.118,Z 552.142,A -85,B 0,C 180,E1 -11266.935,E2 -11266.935} C_VEL
LIN {X 0,Y 400.193,Z 537.834,A -85,B 0,C 180,E1 -11267.922,E2 -11267.922} C_VEL
LIN {X 0,Y 398.317,Z 526.215,A -85,B 0,C 180,E1 -11268.621,E2 -11268.621} C_VEL
LIN {X 0,Y 396.445,Z 517.8,A -85,B 0,C 180,E1 -11269.078,E2 -11269.078} C_VEL
LIN {X 0,Y 396.828,Z 510.177,A -85,B 0,C 180,E1 -11272.382,E2 -11272.382} C_VEL
LIN {X 0,Y 397.48,Z 501.811,A -85,B 0,C 180,E1 -11276.234,E2 -11276.234} C_VEL
LIN {X 0,Y 398.108,Z 495.049,A -85,B 0,C 180,E1 -11279.624,E2 -11279.624} C_VEL
LIN {X 0,Y 398.781,Z 490.29,A -85,B 0,C 180,E1 -11282.227,E2 -11282.227} C_VEL
LIN {X 0,Y 399.297,Z 486.871,A -85,B 0,C 180,E1 -11284.28,E2 -11284.28} C_VEL
LIN {X 0,Y 399.638,Z 483.301,A -85,B 0,C 180,E1 -11286.721,E2 -11286.721} C_VEL
LIN {X 0,Y 399.605,Z 481.691,A -85,B 0,C 180,E1 -11287.993,E2 -11287.993} C_VEL
LIN {X 0,Y 399.168,Z 478.74,A -85,B 0,C 180,E1 -11290.792,E2 -11290.792} C_VEL
LIN {X 0,Y 398.78,Z 476.439,A -85,B 0,C 180,E1 -11293.733,E2 -11293.733} C_VEL
LIN {X 0,Y 398.495,Z 474.968,A -85,B 0,C 180,E1 -11296.542,E2 -11296.542} C_VEL
LIN {X 0,Y 398.316,Z 474.174,A -85,B 0,C 180,E1 -11299.35,E2 -11299.35} C_VEL
LIN {X 0,Y 398.187,Z 473.984,A -85,B 0,C 180,E1 -11302.585,E2 -11302.585} C_VEL
LIN {X 0,Y 397.971,Z 474.445,A -85,B 0,C 180,E1 -11305.59,E2 -11305.59} C_VEL
LIN {X 0,Y 397.753,Z 475.182,A -85,B 0,C 180,E1 -11308.009,E2 -11308.009} C_VEL
LIN {X 0,Y 397.323,Z 476.688,A -85,B 0,C 180,E1 -11311.472,E2 -11311.472} C_VEL
LIN {X 0,Y 397.073,Z 478.538,A -85,B 0,C 180,E1 -11314.863,E2 -11314.863} C_VEL
LIN {X 0,Y 396.792,Z 480.662,A -85,B 0,C 180,E1 -11318.164,E2 -11318.164} C_VEL
LIN {X 0,Y 396.694,Z 482.729,A -85,B 0,C 180,E1 -11321.086,E2 -11321.086} C_VEL
LIN {X 0,Y 401.52,Z 496.964,A -85,B 0,C 180,E1 -11322.13,E2 -11322.13} C_VEL
LIN {X 0,Y 403.123,Z 504.019,A -85,B 0,C 180,E1 -11322.68,E2 -11322.68} C_VEL
LIN {X 0,Y 402.214,Z 517.288,A -85,B 0,C 180,E1 -11323.635,E2 -11323.635} C_VEL
LIN {X 0,Y 401.283,Z 528.081,A -85,B 0,C 180,E1 -11324.615,E2 -11324.615} C_VEL
LIN {X 0,Y 400.237,Z 538.362,A -85,B 0,C 180,E1 -11325.769,E2 -11325.769} C_VEL
LIN {X 0,Y 399.317,Z 547.551,A -85,B 0,C 180,E1 -11327.033,E2 -11327.033} C_VEL
LIN {X 0,Y 398.365,Z 556.537,A -85,B 0,C 180,E1 -11328.552,E2 -11328.552} C_VEL
LIN {X 0,Y 397.725,Z 563.789,A -85,B 0,C 180,E1 -11330.079,E2 -11330.079} C_VEL
LIN {X 0,Y 397.042,Z 570.505,A -85,B 0,C 180,E1 -11331.859,E2 -11331.859} C_VEL
LIN {X 0,Y 396.667,Z 574.351,A -85,B 0,C 180,E1 -11333.174,E2 -11333.174} C_VEL
LIN {X 0,Y 396.362,Z 578.241,A -85,B 0,C 180,E1 -11334.914,E2 -11334.914} C_VEL
LIN {X 0,Y 396.276,Z 579.873,A -85,B 0,C 180,E1 -11335.932,E2 -11335.932} C_VEL
LIN {X 0,Y 396.029,Z 581.936,A -85,B 0,C 180,E1 -11337.966,E2 -11337.966} C_VEL
LIN {X 0,Y 395.941,Z 582.353,A -85,B 0,C 180,E1 -11338.983,E2 -11338.983} C_VEL
LIN {X 0,Y 395.888,Z 582.335,A -85,B 0,C 180,E1 -11340,E2 -11340} C_VEL
LIN {X 0,Y 395.967,Z 581.106,A -85,B 0,C 180,E1 -11342.035,E2 -11342.035} C_VEL
LIN {X 0,Y 396.058,Z 579.848,A -85,B 0,C 180,E1 -11343.052,E2 -11343.052} C_VEL
LIN {X 0,Y 396.062,Z 577.176,A -85,B 0,C 180,E1 -11344.58,E2 -11344.58} C_VEL
LIN {X 0,Y 396.302,Z 573.462,A -85,B 0,C 180,E1 -11346.108,E2 -11346.108} C_VEL
LIN {X 0,Y 396.548,Z 568.613,A -85,B 0,C 180,E1 -11347.639,E2 -11347.639} C_VEL
LIN {X 0,Y 397.026,Z 561.345,A -85,B 0,C 180,E1 -11349.424,E2 -11349.424} C_VEL
LIN {X 0,Y 397.561,Z 553.465,A -85,B 0,C 180,E1 -11350.955,E2 -11350.955} C_VEL
LIN {X 0,Y 398.254,Z 543.643,A -85,B 0,C 180,E1 -11352.485,E2 -11352.485} C_VEL
LIN {X 0,Y 399.052,Z 533.545,A -85,B 0,C 180,E1 -11353.755,E2 -11353.755} C_VEL
LIN {X 0,Y 399.705,Z 521.922,A -85,B 0,C 180,E1 -11354.931,E2 -11354.931} C_VEL
LIN {X 0,Y 400.444,Z 509.613,A -85,B 0,C 180,E1 -11355.916,E2 -11355.916} C_VEL
LIN {X 0,Y 400.858,Z 500.465,A -85,B 0,C 180,E1 -11356.5,E2 -11356.5} C_VEL
LIN {X 0,Y 398.077,Z 487.52,A -85,B 0,C 180,E1 -11357.249,E2 -11357.249} C_VEL
LIN {X 0,Y 396.039,Z 478.229,A -85,B 0,C 180,E1 -11357.692,E2 -11357.692} C_VEL
LIN {X 0,Y 396.06,Z 475.009,A -85,B 0,C 180,E1 -11360.787,E2 -11360.787} C_VEL
LIN {X 0,Y 396.118,Z 471.665,A -85,B 0,C 180,E1 -11364.084,E2 -11364.084} C_VEL
LIN {X 0,Y 396.283,Z 468.297,A -85,B 0,C 180,E1 -11367.459,E2 -11367.459} C_VEL
LIN {X 0,Y 396.296,Z 467.18,A -85,B 0,C 180,E1 -11368.609,E2 -11368.609} C_VEL
LIN {X 0,Y 396.654,Z 467.079,A -85,B 0,C 180,E1 -11372.11,E2 -11372.11} C_VEL
LIN {X 0,Y 397.01,Z 467.031,A -85,B 0,C 180,E1 -11375.481,E2 -11375.481} C_VEL
LIN {X 0,Y 397.129,Z 467.016,A -85,B 0,C 180,E1 -11378.861,E2 -11378.861} C_VEL
LIN {X 0,Y 397.076,Z 467.026,A -85,B 0,C 180,E1 -11382.267,E2 -11382.267} C_VEL
LIN {X 0,Y 397.093,Z 467.02,A -85,B 0,C 180,E1 -11385.069,E2 -11385.069} C_VEL
LIN {X 0,Y 397.071,Z 467.025,A -85,B 0,C 180,E1 -11388.021,E2 -11388.021} C_VEL
LIN {X 0,Y 397.138,Z 467.014,A -85,B 0,C 180,E1 -11391.138,E2 -11391.138} C_VEL
LIN {X 0,Y 397.124,Z 467.018,A -85,B 0,C 180,E1 -11394.497,E2 -11394.497} C_VEL
LIN {X 0,Y 397.083,Z 467.025,A -85,B 0,C 180,E1 -11397.929,E2 -11397.929} C_VEL
LIN {X 0,Y 397.127,Z 467.017,A -85,B 0,C 180,E1 -11401.457,E2 -11401.457} C_VEL
LIN {X 0,Y 397.157,Z 467.014,A -85,B 0,C 180,E1 -11404.488,E2 -11404.488} C_VEL
LIN {X 0,Y 397.113,Z 467.016,A -85,B 0,C 180,E1 -11407.086,E2 -11407.086} C_VEL
LIN {X 0,Y 397.153,Z 467.015,A -85,B 0,C 180,E1 -11410.353,E2 -11410.353} C_VEL
LIN {X 0,Y 397.172,Z 467.012,A -85,B 0,C 180,E1 -11413.553,E2 -11413.553} C_VEL
LIN {X 0,Y 397.234,Z 467.003,A -85,B 0,C 180,E1 -11416.703,E2 -11416.703} C_VEL
LIN {X 0,Y 397.222,Z 467.006,A -85,B 0,C 180,E1 -11419.809,E2 -11419.809} C_VEL
LIN {X 0,Y 397.37,Z 466.986,A -85,B 0,C 180,E1 -11422.888,E2 -11422.888} C_VEL
LIN {X 0,Y 397.259,Z 467,A -85,B 0,C 180,E1 -11424.925,E2 -11424.925} C_VEL
LIN {X 0,Y 397.454,Z 466.978,A -85,B 0,C 180,E1 -11427.973,E2 -11427.973} C_VEL
LIN {X 0,Y 397.585,Z 466.963,A -85,B 0,C 180,E1 -11430,E2 -11430} C_VEL
LIN {X 0,Y 397.38,Z 466.983,A -85,B 0,C 180,E1 -11433.041,E2 -11433.041} C_VEL
LIN {X 0,Y 397.35,Z 466.99,A -85,B 0,C 180,E1 -11436.092,E2 -11436.092} C_VEL
LIN {X 0,Y 397.241,Z 467.002,A -85,B 0,C 180,E1 -11439.162,E2 -11439.162} C_VEL
LIN {X 0,Y 397.224,Z 467.006,A -85,B 0,C 180,E1 -11442.258,E2 -11442.258} C_VEL
LIN {X 0,Y 397.185,Z 467.009,A -85,B 0,C 180,E1 -11445.392,E2 -11445.392} C_VEL
LIN {X 0,Y 397.167,Z 467.012,A -85,B 0,C 180,E1 -11448.573,E2 -11448.573} C_VEL
LIN {X 0,Y 397.101,Z 467.022,A -85,B 0,C 180,E1 -11451.818,E2 -11451.818} C_VEL
LIN {X 0,Y 397.086,Z 467.02,A -85,B 0,C 180,E1 -11452.322,E2 -11452.322} C_VEL
LIN {X 0,Y 396.442,Z 467.102,A -85,B 0,C 180,E1 -11453.168,E2 -11453.168} C_VEL
LIN {X 0,Y 393.645,Z 467.45,A -85,B 0,C 180,E1 -11454.545,E2 -11454.545} C_VEL
LIN {X 0,Y 391.257,Z 467.749,A -85,B 0,C 180,E1 -11455.657,E2 -11455.657} C_VEL
LIN {X 0,Y 390.211,Z 467.877,A -85,B 0,C 180,E1 -11456.516,E2 -11456.516} C_VEL
LIN {X 0,Y 390.115,Z 467.887,A -85,B 0,C 180,E1 -11456.807,E2 -11456.807} C_VEL
LIN {X 0,Y 390.044,Z 467.9,A -85,B 0,C 180,E1 -11460.3,E2 -11460.3} C_VEL
LIN {X 0,Y 390.073,Z 467.898,A -85,B 0,C 180,E1 -11464.024,E2 -11464.024} C_VEL
LIN {X 0,Y 390.05,Z 467.899,A -85,B 0,C 180,E1 -11467.551,E2 -11467.551} C_VEL
LIN {X 0,Y 390.061,Z 467.895,A -85,B 0,C 180,E1 -11470.821,E2 -11470.821} C_VEL
LIN {X 0,Y 390.059,Z 467.899,A -85,B 0,C 180,E1 -11473.886,E2 -11473.886} C_VEL
LIN {X 0,Y 390.063,Z 467.896,A -85,B 0,C 180,E1 -11476.79,E2 -11476.79} C_VEL
LIN {X 0,Y 390.06,Z 467.898,A -85,B 0,C 180,E1 -11479.56,E2 -11479.56} C_VEL
LIN {X 0,Y 390.044,Z 467.897,A -85,B 0,C 180,E1 -11482.45,E2 -11482.45} C_VEL
LIN {X 0,Y 389.957,Z 467.908,A -85,B 0,C 180,E1 -11484.779,E2 -11484.779} C_VEL
LIN {X 0,Y 389.693,Z 467.946,A -85,B 0,C 180,E1 -11487.955,E2 -11487.955} C_VEL
LIN {X 0,Y 389.309,Z 467.992,A -85,B 0,C 180,E1 -11490.829,E2 -11490.829} C_VEL
LIN {X 0,Y 389.059,Z 468.116,A -85,B 0,C 180,E1 -11493.153,E2 -11493.153} C_VEL
LIN {X 0,Y 388.976,Z 471.904,A -85,B 0,C 180,E1 -11496.578,E2 -11496.578} C_VEL
LIN {X 0,Y 388.987,Z 475.673,A -85,B 0,C 180,E1 -11499.97,E2 -11499.97} C_VEL
LIN {X 0,Y 388.941,Z 478.147,A -85,B 0,C 180,E1 -11502.179,E2 -11502.179} C_VEL
LIN {X 0,Y 392.229,Z 493.668,A -85,B 0,C 180,E1 -11502.967,E2 -11502.967} C_VEL
LIN {X 0,Y 393.883,Z 501.758,A -85,B 0,C 180,E1 -11503.478,E2 -11503.478} C_VEL
LIN {X 0,Y 393.189,Z 513.926,A -85,B 0,C 180,E1 -11504.315,E2 -11504.315} C_VEL
LIN {X 0,Y 392.58,Z 525.589,A -85,B 0,C 180,E1 -11505.34,E2 -11505.34} C_VEL
LIN {X 0,Y 391.793,Z 536.345,A -85,B 0,C 180,E1 -11506.514,E2 -11506.514} C_VEL
LIN {X 0,Y 391.022,Z 545.977,A -85,B 0,C 180,E1 -11507.808,E2 -11507.808} C_VEL
LIN {X 0,Y 390.455,Z 553.959,A -85,B 0,C 180,E1 -11509.106,E2 -11509.106} C_VEL
LIN {X 0,Y 389.9,Z 561.814,A -85,B 0,C 180,E1 -11510.664,E2 -11510.664} C_VEL
LIN {X 0,Y 389.483,Z 568.097,A -85,B 0,C 180,E1 -11512.222,E2 -11512.222} C_VEL
LIN {X 0,Y 389.241,Z 573.099,A -85,B 0,C 180,E1 -11513.78,E2 -11513.78} C_VEL
LIN {X 0,Y 388.988,Z 576.955,A -85,B 0,C 180,E1 -11515.336,E2 -11515.336} C_VEL
LIN {X 0,Y 388.974,Z 579.757,A -85,B 0,C 180,E1 -11516.893,E2 -11516.893} C_VEL
LIN {X 0,Y 388.891,Z 581.093,A -85,B 0,C 180,E1 -11517.928,E2 -11517.928} C_VEL
LIN {X 0,Y 388.807,Z 582.003,A -85,B 0,C 180,E1 -11518.964,E2 -11518.964} C_VEL
LIN {X 0,Y 388.8,Z 582.474,A -85,B 0,C 180,E1 -11520,E2 -11520} C_VEL
LIN {X 0,Y 388.842,Z 582.55,A -85,B 0,C 180,E1 -11521.035,E2 -11521.035} C_VEL
LIN {X 0,Y 388.94,Z 582.23,A -85,B 0,C 180,E1 -11522.071,E2 -11522.071} C_VEL
LIN {X 0,Y 389.058,Z 581.458,A -85,B 0,C 180,E1 -11523.106,E2 -11523.106} C_VEL
LIN {X 0,Y 389.222,Z 580.28,A -85,B 0,C 180,E1 -11524.142,E2 -11524.142} C_VEL
LIN {X 0,Y 389.245,Z 577.741,A -85,B 0,C 180,E1 -11525.699,E2 -11525.699} C_VEL
LIN {X 0,Y 389.76,Z 573.844,A -85,B 0,C 180,E1 -11527.368,E2 -11527.368} C_VEL
LIN {X 0,Y 390.179,Z 569.456,A -85,B 0,C 180,E1 -11528.807,E2 -11528.807} C_VEL
LIN {X 0,Y 390.837,Z 563.555,A -85,B 0,C 180,E1 -11530.359,E2 -11530.359} C_VEL
LIN {X 0,Y 391.566,Z 556.198,A -85,B 0,C 180,E1 -11531.912,E2 -11531.912} C_VEL
LIN {X 0,Y 392.389,Z 548.722,A -85,B 0,C 180,E1 -11533.201,E2 -11533.201} C_VEL
LIN {X 0,Y 393.336,Z 539.707,A -85,B 0,C 180,E1 -11534.486,E2 -11534.486} C_VEL
LIN {X 0,Y 394.52,Z 528.447,A -85,B 0,C 180,E1 -11535.789,E2 -11535.789} C_VEL
LIN {X 0,Y 395.66,Z 516.298,A -85,B 0,C 180,E1 -11536.91,E2 -11536.91} C_VEL
LIN {X 0,Y 396.517,Z 505.872,A -85,B 0,C 180,E1 -11537.673,E2 -11537.673} C_VEL
LIN {X 0,Y 394.94,Z 498.259,A -85,B 0,C 180,E1 -11538.281,E2 -11538.281} C_VEL
LIN {X 0,Y 391.107,Z 486.479,A -85,B 0,C 180,E1 -11539.207,E2 -11539.207} C_VEL
LIN {X 0,Y 389.578,Z 482.035,A -85,B 0,C 180,E1 -11539.53,E2 -11539.53} C_VEL
LIN {X 0,Y 389.601,Z 477.974,A -85,B 0,C 180,E1 -11543.382,E2 -11543.382} C_VEL
LIN {X 0,Y 389.722,Z 474.382,A -85,B 0,C 180,E1 -11546.797,E2 -11546.797} C_VEL
LIN {X 0,Y 389.794,Z 470.614,A -85,B 0,C 180,E1 -11550.321,E2 -11550.321} C_VEL
LIN {X 0,Y 389.785,Z 468.119,A -85,B 0,C 180,E1 -11552.746,E2 -11552.746} C_VEL
LIN {X 0,Y 389.991,Z 467.909,A -85,B 0,C 180,E1 -11555.812,E2 -11555.812} C_VEL
LIN {X 0,Y 390.072,Z 467.897,A -85,B 0,C 180,E1 -11559.218,E2 -11559.218} C_VEL
LIN {X 0,Y 390.047,Z 467.902,A -85,B 0,C 180,E1 -11562.374,E2 -11562.374} C_VEL
LIN {X 0,Y 390.049,Z 467.901,A -85,B 0,C 180,E1 -11565.355,E2 -11565.355} C_VEL
LIN {X 0,Y 390.121,Z 468.062,A -85,B 0,C 180,E1 -11566.672,E2 -11566.672} C_VEL
LIN {X 0,Y 391.103,Z 473.547,A -85,B 0,C 180,E1 -11569.691,E2 -11569.691} C_VEL
LIN {X 0,Y 392.166,Z 480.055,A -85,B 0,C 180,E1 -11573.105,E2 -11573.105} C_VEL
LIN {X 0,Y 392.147,Z 483.896,A -85,B 0,C 180,E1 -11575.005,E2 -11575.005} C_VEL
LIN {X 0,Y 391.392,Z 491.518,A -85,B 0,C 180,E1 -11578.618,E2 -11578.618} C_VEL
LIN {X 0,Y 390.75,Z 499.114,A -85,B 0,C 180,E1 -11582.119,E2 -11582.119} C_VEL
LIN {X 0,Y 390.145,Z 506.689,A -85,B 0,C 180,E1 -11585.524,E2 -11585.524} C_VEL
LIN {X 0,Y 389.641,Z 514.229,A -85,B 0,C 180,E1 -11588.854,E2 -11588.854} C_VEL
LIN {X 0,Y 389.42,Z 518.875,A -85,B 0,C 180,E1 -11590.804,E2 -11590.804} C_VEL
LIN {X 0,Y 392.116,Z 532.418,A -85,B 0,C 180,E1 -11591.601,E2 -11591.601} C_VEL
LIN {X 0,Y 393.539,Z 547.081,A -85,B 0,C 180,E1 -11592.6,E2 -11592.6} C_VEL
LIN {X 0,Y 393.916,Z 555.682,A -85,B 0,C 180,E1 -11593.281,E2 -11593.281} C_VEL
LIN {X 0,Y 392.835,Z 567.354,A -85,B 0,C 180,E1 -11594.3,E2 -11594.3} C_VEL
LIN {X 0,Y 391.826,Z 577.988,A -85,B 0,C 180,E1 -11595.457,E2 -11595.457} C_VEL
LIN {X 0,Y 390.966,Z 587.76,A -85,B 0,C 180,E1 -11596.75,E2 -11596.75} C_VEL
LIN {X 0,Y 390.11,Z 597.382,A -85,B 0,C 180,E1 -11598.307,E2 -11598.307} C_VEL
LIN {X 0,Y 389.499,Z 605.159,A -85,B 0,C 180,E1 -11599.867,E2 -11599.867} C_VEL
LIN {X 0,Y 389.091,Z 612.412,A -85,B 0,C 180,E1 -11601.692,E2 -11601.692} C_VEL
LIN {X 0,Y 388.906,Z 617.643,A -85,B 0,C 180,E1 -11603.254,E2 -11603.254} C_VEL
LIN {X 0,Y 388.837,Z 621.673,A -85,B 0,C 180,E1 -11604.815,E2 -11604.815} C_VEL
LIN {X 0,Y 388.747,Z 623.718,A -85,B 0,C 180,E1 -11605.853,E2 -11605.853} C_VEL
LIN {X 0,Y 388.78,Z 625.335,A -85,B 0,C 180,E1 -11606.891,E2 -11606.891} C_VEL
LIN {X 0,Y 388.847,Z 626.53,A -85,B 0,C 180,E1 -11607.928,E2 -11607.928} C_VEL
LIN {X 0,Y 388.81,Z 627.253,A -85,B 0,C 180,E1 -11608.964,E2 -11608.964} C_VEL
LIN {X 0,Y 388.81,Z 627.55,A -85,B 0,C 180,E1 -11610,E2 -11610} C_VEL
LIN {X 0,Y 388.801,Z 627.436,A -85,B 0,C 180,E1 -11611.036,E2 -11611.036} C_VEL
LIN {X 0,Y 388.845,Z 626.913,A -85,B 0,C 180,E1 -11612.072,E2 -11612.072} C_VEL
